# B&R Automation Studio project TD52 (part 102)

#### perm_par.var
```iecst
VAR
	tParaIntern : ParaHandler_typ; (*Connector type to perm_par*)
	tMM2ParaBase_ReadBack : MM2ParaBase_type; (*INTERNAL! V4.06 new readback structure for information from previous tasks*)
	bWriteDataObj : BOOL; (* TRUE=write data object module *)
	bDataObjLenErr : BOOL; (*Error occured in permem: data module size missmatch*)
	bCreateDataObj : BOOL; (* TRUE=create new data object *)
	bWriteOnce : BOOL; (* write permanent memory once *)
	DatObjCreate_01 : DatObjCreate; (* data object create *)
	DatObjInfoBak_02 : DatObjInfo; (* data object info *)
	DatObjDelete_01 : DatObjDelete; (* data object delete *)
	DatObjRead_01 : DatObjRead; (* data object read *)
	DatObjRead_02 : DatObjRead; (* manual initiated data object read *)
	DatObjWrite_01 : DatObjWrite; (* data object write *)
	DatObjDelete_02 : DatObjDelete; (* data object delete *)
	DatObjDelete_11 : DatObjDelete; (*Delete Backup File*)
	DatObjInfo_01 : DatObjInfo; (* data object info *)
	DatObjInfo_02 : DatObjInfo; (* data object info *)
	szModuleName : STRING[35]; (* module name of object *)
	szModuleNameBackup : STRING[35]; (* module name of posiibly created backup object *)
	DatObjCopy_01 : DatObjCopy;
	bCopyDataObj : BOOL;
	TON_WarnDelay : TON;
	TON_WritePMEM : TON; (* delay write permanent memory *)
	ulPMPointer : UDINT; (* adress of actual checksum value *)
	ulChecksum : UDINT; (* parameter checksum value *)
	pm_len : UDINT; (* permanent value lenght *)
	ulChecksumOld : UDINT; (* last vlaue of parameter checksum *)
	ulChkValue : UDINT; (* actual value of parameter pointer *)
	pm_id : UDINT; (* permanent value identifier *)
	pm_p : UDINT; (* permanent value pointer *)
	DatObjInfo_META : DatObjInfo;
	DatObjRead_META : DatObjRead;
	szMetaDataRaw : STRING[2000];
	szMetaData : ARRAY[0..4] OF STRING[35];
	szMetaDataVis : ARRAY[0..3] OF STRING[35];
	ssIndex : INT;
	ssCount : INT;
	ucMetaDataRaw : ARRAY[0..2000] OF USINT;
	ssCount2 : INT;
	szMetaDataFile : STRING[10];
	szText1 : STRING[20];
	pv_adr_IN_XX_tPB2MM : UDINT;
	pv_lng : UDINT;
	pv_lng_IN_XX_tPB2MM : UDINT;
	pv_lng_OUT_XX_tPB2MM : UDINT;
	szText2 : STRING[20];
	pv_adr_OUT_XX_tXX2PB : UDINT;
END_VAR
VAR CONSTANT
	ERR_NOERROR : UINT := 0;
END_VAR
VAR
	usPMWriteCnt : UINT;
	pm_Error : UDINT; (* permanent value error *) (* Deleted: pm : ParaMem_typ; permanent memory tags mathias, 22.8.11*)
	fun_Error : UDINT := 0; (*state > 0 = function error*)
	xLocalParaCheck : ParaCheckFUB; (*local function instance to check parameter values*)
	TON_ParaSetupOk : TON;
	bParaCheckSystemOk : BOOL;
	iDebug_ParaOkChecked : UDINT;
	bRestoreBackupDataObj : BOOL := FALSE;
	bRestoreDataObjContent : BOOL := FALSE;
	pm_id_backup : UDINT;
	pm_p_Backup : UDINT;
	DatObjCopy_02 : DatObjCopy;
	bDeleteBackupDataObj : BOOL := FALSE; (*Command to delete backup data module file on purpose*)
	bDebugPara : ARRAY[0..5] OF BOOL;
	ssIndex2 : INT;
	ssIndex3 : INT;
	ssIndex4 : INT;
	ssIndexVis : INT;
	szText : STRING[40];
	pv_adr_Para : UDINT;
	szParaSnippet : ARRAY[0..5] OF STRING[150];
	szParaIndex : STRING[10];
	slValue : DINT;
	iModuleDLD_ResetCount : INT;
	bDownloadDetected : BOOL;
	bFlagParaStructCopyWorking : BOOL; (*true, if cyclic para copying is active, 1 false cycle at every copy *)
	bStoreInitParaInDataObj : BOOL := FALSE;
	bTestflag : BOOL;
	bReadOutMETA_Once : BOOL;
	tParaCheck_iPvAdress : ARRAY[0..5] OF UDINT;
	tParaCheck_iPvLengt : ARRAY[0..5] OF UDINT;
	tParaCheck_rPvValue : ARRAY[0..5] OF REAL;
	tParaCheck_rRangeMIN : ARRAY[0..5] OF REAL;
	tParaCheck_rRangeMAX : ARRAY[0..5] OF REAL;
	tParaCheck_szPvName : ARRAY[0..5] OF STRING[35];
	ssFormatDetected : INT;
	szMetaDataPart : STRING[150];
	szFullTaskName : STRING[35];
	szFullMetaModuleName : STRING[35];
	debugLen : INT;
	debugSize : INT := 0;
	strcat_adr1 : UDINT;
	strcat_adr2 : UDINT;
	ssIndexTN : INT;
	bAlternate : BOOL;
	n : INT;
	iAlternateChecksum : DINT;
	iAlternateChecksumOld : DINT;
	ulDebugChkValue : ARRAY[0..999] OF UDINT;
	Adr1 : UDINT;
	Adr2 : UDINT;
	usPMWriteCntStepsize : UINT := 1; (*different step sizes to help debug*)
	usPMWriteCntXOR : UINT;
	usPMWriteCntAltSum : UINT;
	ulAdrPM : UDINT;
	usChkValuePM : USINT;
	ulAdrPara : UDINT;
	ulPara_len : UDINT;
	usChkValuePara : USINT;
	iDebugCountPMDifferences : DINT := 0;
	bEngineRunDetected : BOOL; (*detection status bit autocommand 100 /101  for engine run state*)
	ucMetaDataDebugInfoLine : ARRAY[0..24] OF STRING[80];
	ssIndexMand : INT := 0;
	szMetaDataMand : STRING[35];
	iMyErrorInfo_Autoreset : DINT; (*internal autoreset counter*)
	ssIndex_Version : INT; (*internal*)
	ssIndex_BU : INT; (*internal*)
	ssIndex_BU2 : INT; (*internal*)
END_VAR
```

### Program Logical/Generator/VisGC (IEC, version 4.09.0) - Visualization <-> Metamodule

#### VisGCCyclic.st
```iecst
(********************************************************************
VisGC	 			 General issues are handled here

This code is confidential and proprietary to the INNIO Company.
It may not be used in any form, or reproduced in any manner,
without written permission of the INNIO Company.
Copyright, INNIO Company, 2019

Customized modifications: -
------------------------

History:
-------
4.00.0	01.01.2013	ganguly		new
4.00.0	16.05.2014	lettenb.	cleanup
4.04.0	29.06.2016	lettenb.	tGen_T_In2 added, Dig142
4.05.0	30.11.2017	lettenb.	Q-management, unused MM2VIS-var removed
4.07.0	11.10.2018	lettenb.	Di: tU_Gen_Inc/Dec added for diagnosis
		29.04.2019	lettenb.	bU_Gen_Inc/Dec puls elongation for vis added(request requisition, mayer)
4.09.0	02.12.2019	lettenb.	ground failure counter added

Instructions for use: -
--------------------

Outstandings:
------------

*******************************************************************************)

PROGRAM _CYCLIC

	MM2VIS.bP_CosPCtr_Red_F_Hi     := OUT_GC.bP_Red_CosPCtr_F_Hi;
	MM2VIS.bP_CosPCtr_Red_F_Lo     := OUT_GC.bP_Red_CosPCtr_F_Lo;
	MM2VIS.bP_CosPCtr_Red_U_Hi     := OUT_GC.bP_Red_CosPCtr_U_Hi;
	MM2VIS.bP_CosPCtr_Red_U_Lo     := OUT_GC.bP_Red_CosPCtr_U_Lo;
	MM2VIS.rP_Gen_ppt              := rP_Gen_ppt;

	MM2VIS.rPF_CosPCtr_Set_Ctr13   := rPF_CosPCtr_Set_Ctr13;
	MM2VIS.rP_Red_CosPCtr_F        := rP_CosPCtr_F_Red;
	MM2VIS.rP_Red_CosPCtr_U        := rP_CosPCtr_U_Red;
	MM2VIS.rP_Red_CosPCtr_T        := rP_CosPCtr_T_Red;

	MM2VIS.rQ_CosPCtr_Set          := rQ_CosPCtr_Set;

	MM2VIS.rU_Gen_Exc              := OUT_GC.rU_Gen_Exc;

	MM2VIS.rT_Gen_Bear_A_Act       := IN_GC.tT_Gen_Bear_A_Act.Ai;
	MM2VIS.rT_Gen_Bear_B_Act       := IN_GC.tT_Gen_Bear_B_Act.Ai;
	MM2VIS.rT_Gen_Wind_Act_L1      := IN_GC.tT_Gen_Wind_Act_L1.Ai;
	MM2VIS.rT_Gen_Wind_Act_L2      := IN_GC.tT_Gen_Wind_Act_L2.Ai;
	MM2VIS.rT_Gen_Wind_Act_L3      := IN_GC.tT_Gen_Wind_Act_L3.Ai;
	MM2VIS.rT_Gen_Wind_Act         := IN_GC.tT_Gen_Wind.Ai;

	(* Oilskid *)
	MM2VIS.bOilSkid_PumpLP_Dem 		:= OUT_GC.tOilSkid_PumpLP.Do;
	MM2VIS.bOilSkid_PumpHP_Dem		:= OUT_GC.tOilSkid_PumpHP.Do OR OUT_GC.tOilSkid_PumpHP_UPS.Do;
	MM2VIS.bOilSkid_PumpC_Dem 		:= OUT_GC.tOilSkid_PumpC.Do;
	MM2VIS.bOilSkid_Fan_Dem 		:= OUT_GC.tOilSkid_Fan.Do;
	MM2VIS.bOilSkid_Heater_Dem 		:= OUT_GC.tOilSkid_Heater.Do;
	MM2VIS.rLev_OilSkid_Tank		:= IN_GC.tLev_OilSkid_Tank.Ai;
	MM2VIS.rT_OilSkid_Tank			:= IN_GC.tT_OilSkid_Tank.Ai;
	MM2VIS.rPr_OilSkid_HP_NDE		:= IN_GC.tPr_OilSkid_HP_NDE.Ai;
	MM2VIS.rPr_OilSkid_HP_DE		:= IN_GC.tPr_OilSkid_HP_DE.Ai;
	MM2VIS.rFlow_OilSkid_DE			:= IN_GC.tFlow_OilSkid_DE.Ai;
	MM2VIS.rFlow_OilSkid_NDE		:= IN_GC.tFlow_OilSkid_NDE.Ai;
	MM2VIS.rT_OilSkid_Supply		:= IN_GC.tT_OilSkid_Supply.Ai;

	MM2VIS.rF_GenBear_DE1			:= IN_GC.tF_GenBear_DE1.Ai;
	MM2VIS.rF_GenBear_DE2			:= IN_GC.tF_GenBear_DE2.Ai;
	MM2VIS.rF_GenBear_NDE1			:= IN_GC.tF_GenBear_NDE1.Ai;
	MM2VIS.rF_GenBear_NDE2			:= IN_GC.tF_GenBear_NDE2.Ai;

	MM2VIS.rGen_T_In				:= IN_GC.tGen_T_In.Ai;
	MM2VIS.rGen_T_In2				:= IN_GC.tGen_T_In2.Ai;
	MM2VIS.rT_GenAirOut				:= IN_GC.tT_GenAirOut.Ai;

	xTP_U_Gen_Inc(IN:= EDGEPOS(IN_GC.tU_Gen_Inc.Di OR IN_GC.tU_Adj_Plus.Di), PT:= T#2s);(* DI voltage adjustment external (increasing)*)
	MM2VIS.bU_Gen_Inc				:= xTP_U_Gen_Inc.Q;

	xTP_U_Gen_Dec(IN:= EDGEPOS(IN_GC.tU_Gen_Dec.Di OR IN_GC.tU_Adj_Minus.Di), PT:= T#2s);(* DI voltage adjustment external (decreasing)*)
	MM2VIS.bU_Gen_Dec				:= xTP_U_Gen_Dec.Q;

	MM2VIS.bCntGndFail_Visible 		:= IN_GC.tGndFaultW.GoodQual; (* counter visibility *)

END_PROGRAM
```

#### VisGC.var
```iecst
VAR
  	xTP_U_Gen_Inc : TP;
  	xTP_U_Gen_Dec : TP;
END_VAR

VAR CONSTANT

END_VAR
```

### Program Logical/Generator/MMUEarthFault (IEC) - MMU Earth Fault detection

#### MMUEarthFaultCyclic.st - Program
```iecst
(********************************************************************
MMUEarthFault	 			 Earth Fault Detection via MMU Signals

This code is confidential and proprietary to the INNIO Company.
It may not be used in any form, or reproduced in any manner,
without written permission of the INNIO Company.
Copyright, INNIO Company, 2023

Customized modifications: -
------------------------

History:
-------
4.13.0	29.06.2023	Perktold	new

Instructions for use: -
--------------------

Outstandings:
------------

*******************************************************************************)
PROGRAM _CYCLIC

IF Para.rU_Gen_Nom[1] <> 0 THEN

	//Activate monitoring 2s after at least one Ph-Ph-Voltage exceeds 50% nominal voltage
	xTON_MonAct(IN := (MAX(IN_GC.tU_L1L2[1].Ai, IN_GC.tU_L2L3[1].Ai, IN_GC.tU_L3L1[1].Ai) > (Para.rU_Gen_Nom[1] * 0.5)), PT := T#2s);

	IF xTON_MonAct.Q THEN

		//Read pos. zero crossing time stamps and convert to [ms]
		rTimeStamp_PosZeroCrossing_UGen1 := DINT_TO_REAL(IN_GC.iTimeStamp_PosZeroCrossing_UGen1) / 4096000;	(* [ms] *)
		rTimeStamp_PosZeroCrossing_UGen2 := DINT_TO_REAL(IN_GC.iTimeStamp_PosZeroCrossing_UGen2) / 4096000;	(* [ms] *)
		rTimeStamp_PosZeroCrossing_UGen3 := DINT_TO_REAL(IN_GC.iTimeStamp_PosZeroCrossing_UGen3) / 4096000;	(* [ms] *)

		//Correct values for easy comparison if values overrun the DINT the negatve values get corrected by 1048.5759ms (total DINT range)
		iNumNeg	:= 0;
		IF ABS(rTimeStamp_PosZeroCrossing_UGen1) > 200 AND ABS(rTimeStamp_PosZeroCrossing_UGen2) > 200 AND ABS(rTimeStamp_PosZeroCrossing_UGen3) > 200 THEN
			IF rTimeStamp_PosZeroCrossing_UGen1 < 0.0 THEN	iNumNeg	:= iNumNeg + 1;	END_IF;
			IF rTimeStamp_PosZeroCrossing_UGen2 < 0.0 THEN	iNumNeg	:= iNumNeg + 1;	END_IF;
			IF rTimeStamp_PosZeroCrossing_UGen3 < 0.0 THEN	iNumNeg	:= iNumNeg + 1;	END_IF;

			IF (iNumNeg = 1) OR (iNumNeg = 2) THEN
				IF rTimeStamp_PosZeroCrossing_UGen1 < 0.0 THEN
					rTimeStamp_Calc_UGen1	:= rTimeStamp_PosZeroCrossing_UGen1 + 1048.57599975586;	(* [ms] *)
				ELSE
					rTimeStamp_Calc_UGen1	:= rTimeStamp_PosZeroCrossing_UGen1;					(* [ms] *)
				END_IF;

				IF rTimeStamp_PosZeroCrossing_UGen2 < 0.0 THEN
					rTimeStamp_Calc_UGen2	:= rTimeStamp_PosZeroCrossing_UGen2 + 1048.57599975586;	(* [ms] *)
				ELSE
					rTimeStamp_Calc_UGen2	:= rTimeStamp_PosZeroCrossing_UGen2;					(* [ms] *)
				END_IF;

				IF rTimeStamp_PosZeroCrossing_UGen3 < 0.0 THEN
					rTimeStamp_Calc_UGen3	:= rTimeStamp_PosZeroCrossing_UGen3 + 1048.57599975586;	(* [ms] *)
				ELSE
					rTimeStamp_Calc_UGen3	:= rTimeStamp_PosZeroCrossing_UGen3;					(* [ms] *)
				END_IF;
			ELSE
				rTimeStamp_Calc_UGen1	:= rTimeStamp_PosZeroCrossing_UGen1;						(* [ms] *)
				rTimeStamp_Calc_UGen2	:= rTimeStamp_PosZeroCrossing_UGen2;						(* [ms] *)
				rTimeStamp_Calc_UGen3	:= rTimeStamp_PosZeroCrossing_UGen3;						(* [ms] *)
			END_IF;
		ELSE
			rTimeStamp_Calc_UGen1	:= rTimeStamp_PosZeroCrossing_UGen1;							(* [ms] *)
			rTimeStamp_Calc_UGen2	:= rTimeStamp_PosZeroCrossing_UGen2;							(* [ms] *)
			rTimeStamp_Calc_UGen3	:= rTimeStamp_PosZeroCrossing_UGen3;							(* [ms] *)
		END_IF;

		//get the three values in the right order
		rTimeStamp_max	:= MAX(rTimeStamp_Calc_UGen1, rTimeStamp_Calc_UGen2, rTimeStamp_Calc_UGen3);
		rTimeStamp_min	:= MIN(rTimeStamp_Calc_UGen1, rTimeStamp_Calc_UGen2, rTimeStamp_Calc_UGen3);

		IF (rTimeStamp_Calc_UGen1 <> rTimeStamp_max) AND (rTimeStamp_Calc_UGen1 <> rTimeStamp_min) THEN
			rTimeStamp_mid	:= rTimeStamp_Calc_UGen1;
		ELSIF (rTimeStamp_Calc_UGen2 <> rTimeStamp_max) AND (rTimeStamp_Calc_UGen2 <> rTimeStamp_min) THEN
			rTimeStamp_mid	:= rTimeStamp_Calc_UGen2;
		ELSE
			rTimeStamp_mid	:= rTimeStamp_Calc_UGen3;
		END_IF;

		//Calculate time difference beween the time stamps
		rDelta_1 := rTimeStamp_mid - rTimeStamp_min;							(* [ms] *)
		rDelta_2 := rTimeStamp_max - rTimeStamp_mid;							(* [ms] *)

		rTPeriodTime	:= 1.0 / LIMIT(0.1, IN_GC.tF_MMD[1].Ai, 70.0) * 1000;	(* [ms] *)
		//convert to angle difference
		rDAng_1			:= rDelta_1 / rTPeriodTime * 360.0;						(* [Deg] *)
		rDAng_2			:= rDelta_2 / rTPeriodTime * 360.0;						(* [Deg] *)

		//Check if the values are 120[Deg] +- rDAng_Dev
		IF (rDAng_1 > (120.0 - rDAng_Dev)) AND (rDAng_1 < (120.0 + rDAng_Dev)) THEN
			bDANg_1_ok	:= TRUE;
		ELSE
			bDANg_1_ok	:= FALSE;
		END_IF

		IF (rDAng_2 > (120.0 - rDAng_Dev)) AND (rDAng_2 < (120.0 + rDAng_Dev)) THEN
			bDANg_2_ok	:= TRUE;
		ELSE
			bDANg_2_ok	:= FALSE;
		END_IF

		//trigger warning and trip if at least on value stays out of range for a vertain time
		xTON_warning(IN := ((NOT bDANg_1_ok OR NOT bDANg_2_ok) AND Para.bMMDGroundFaultMonAct AND (Para.tTi_MMDGroundFaultWarning > T#0ms)), PT := Para.tTi_MMDGroundFaultWarning);
		xTON_trip(IN 	:= ((NOT bDANg_1_ok OR NOT bDANg_2_ok) AND Para.bMMDGroundFaultMonAct AND (Para.tTi_MMDGroundFaultTrip > T#0ms)), PT := Para.tTi_MMDGroundFaultTrip);

		bMsg9372_set			:= xTON_warning.Q;		(*W9372 Multi measurement device: Earth failure generator*)
		bMsg2373_set			:= xTON_trip.Q;			(*A2373 Multi measurement device: Earth failure generator*)
	ELSE
		bMsg9372_set			:= FALSE;
		bMsg2373_set			:= FALSE;
		xTON_warning(IN := FALSE, PT := Para.tTi_MMDGroundFaultWarning);
		xTON_trip(IN 	:= FALSE, PT := Para.tTi_MMDGroundFaultTrip);
	END_IF;
ELSE
	bMsg9372_set	:= FALSE;
	bMsg2373_set	:= FALSE;
	xTON_warning(IN	:= FALSE, PT := Para.tTi_MMDGroundFaultWarning);
	xTON_trip(IN 	:= FALSE, PT := Para.tTi_MMDGroundFaultTrip);
	xTON_MonAct(IN 	:= FALSE, PT := T#2s);
END_IF;

END_PROGRAM
```

#### MMUEarthFault.var - Variables
```iecst
VAR
	rTimeStamp_PosZeroCrossing_UGen1 : REAL := 0.0; (*[ms]*)
	rTimeStamp_PosZeroCrossing_UGen2 : REAL := 0.0; (*[ms]*)
	rTimeStamp_PosZeroCrossing_UGen3 : REAL := 0.0; (*[ms]*)
	rTPeriodTime : REAL; (*[ms]*)
	rTimeStamp_Calc_UGen1 : REAL := 0.0;
	rTimeStamp_Calc_UGen2 : REAL := 0.0;
	rTimeStamp_Calc_UGen3 : REAL := 0.0;
	rTimeStamp_max : REAL := 0.0;
	rTimeStamp_min : REAL := 0.0;
	rTimeStamp_mid : REAL := 0.0;
	iNumNeg : INT := 0;
	rDelta_1 : REAL := 0.0;
	rDelta_2 : REAL := 0.0;
	rDAng_1 : REAL := 0.0;
	rDAng_2 : REAL := 0.0;
	rDAng_Dev : REAL := 10.0;
	bDANg_1_ok : BOOL := 0;
	bDANg_2_ok : BOOL := 0;
	xTON_warning : TON;
	xTON_trip : TON;
	xTON_MonAct : TON;
END_VAR
```

### Package Logical/GasMeteringUnit - GD: Gas Metering Unit Device

### Data object Logical/GasMeteringUnit/META_GD (Simple) - Simple data object.

#### META_GD.dat
```
; *******************************************************************************
; AGGR: Module Meta Data (data module)
;
; This code is confidential and proprietary to the INNIO Company.
; It may not be used in any form, or reproduced in any manner, without the express
; written permission of the INNIO Company.
; Copyright, INNIO Company, 2023
;
; Customized modifications: -
; ------------------------
;
; History:
; -------
; V3.99	06-03-2013	Weitzer, generated for modular software
; V4.00 11-09-2013  pankajrodey, updated file with relevant information
; V4.01 18-10-2013  Zengerer   typo corr., NO duplicate para Chk entries!
; 		08-05-2014  Weitzer, switch to CAN interface identifier from HAL_IO
;							 "hard code" missing parameters
; V4.04.00.00	04-07-2016	Gwiggner,	Bugfix: Tecjet Monitoring
; V4.04.00.00	05-08-2016	Gwiggner,	Bugfix: Mapping bDualTJ
; V4.04.00.00	28-10-2016	Gwiggner,	Bugfix: correction interpolation of gas density
; V4.05.00.00	27.07.2017	Messner,	CAN Diagnosis Picture added
; V4.05.01.00	05.04.2018	Perktold,	GMU - Monitoring Delay for TJs increased from 5 to 7s
; V4.11.00.00	15.11.2021	Perktold,	defined ucTecNr as local variable, correction REAL_TO_USINT -> INT_TO_USINT, A3093 DGS
; V4.12.00.00	13.12.2022	Gwiggner,	GMU self diagnosis
; V4.12.00.00	22.01.2023	Zuschnig,	Interpolation od gas density done in EC module
; V4.13.00.00	16.11.2022	Gwiggner,	adaption for W3213 & B3249
;
; Instructions for use:
; --------------------
; make only changes at the version numbers
;
; Outstandings:
; ------------
;
; *******************************************************************************
;
"<META>"
;
; Module ID
"<MODUL>GD</MODUL>"
;
; Module Version (xx.yy.zz.cc)
"<VERSION>04.13.00.00</VERSION>"
;
; Module Basisupdate Version BU (00-99)
"<BASISUPDATE_VERSION>00</BASISUPDATE_VERSION>"
;
; Optional: specify order number for limitated module usage
"<ORDER></ORDER>" ;<!--(optional for restricted customizations; missing statement makes module valid for all orders)-->
;
; Parameter Check <PARAn Name='aAbcdef' MIN='xxx' MAX='yyy' />  (watch for correct spacings and apostrophs!)
"<PARAMETER_CHK>"
"<PARA1 Name='iEng_Motortype' MIN='208' MAX='920' />"
"<PARA2 Name='iN_GMU_Devices' MIN='0' MAX='5' />"
"<PARA3 Name='usGasDensN[1]' MIN='200' MAX='2500' />"
"<PARA4 />"
"<PARA5 />"
"</PARAMETER_CHK>"
;
; <--Permanent Datamodule Filenames:  NAME ist ohne Dateiendung einzutragen; Nur für Counter und interne Parameter verwenden-->
"<DATAMODULES>" ;<!-- optional; mehrere DATAMODULES erlaubt-->
"	<DATAMODULE>par_GD</DATAMODULE>"
"</DATAMODULES>"
;
; Dependencies Modules (MMxx.yy.zz.cc)
"<DEPENDENCIES>"
"	<DEPENDENCY MODULE='AB' VERSION='04.00.00.00' />"
"	<DEPENDENCY MODULE='PB' VERSION='04.00.00.00' />"
"	<DEPENDENCY MODULE='GT' VERSION='04.12.00.00' />"
"	<DEPENDENCY MODULE='OP' VERSION='04.00.00.00' />"
"	<DEPENDENCY MODULE='HA' VERSION='04.05.00.00' />"
"	<DEPENDENCY MODULE='EC' VERSION='04.12.00.00' />"
"   <DEPENDENCY VISVERSION='02.06.00.00' />"			; Dependencies Visualization
"</DEPENDENCIES>"
;
; Module function description
"<MODULEFUNCTION>" ;<!-- short overview documentation of module function; add reference to detailed information, if available-->
"	<General>	"
"	GD Module for the TecJet(tm) valve actuator - an integrated and digitally compensated control valve and actuator system"
" 	for regulating and metering the flow of gas "
"	</General>	"
""
"	<F1 Name='Gas metering' LastModified='4.0.0.0'>"
"	These paramaeters of the Air-Fuel mixture are measured by the module:	"
"	Valve differential pressure, Valve position, Gas Temperature, Running hours, Software version, Gas pressure	"
"	</F1>"
"	<F2 Name='Errors and alarms' LastModified='4.0.0.0'>"
"	Errors in the Tecjet module are sent by this module to the controller	"
"	</F2>"
"	<F3 Name='enter name of main function 3 here' LastModified='4.0.0.0'>"
"	Enter function 3 description for module here.	"
"	</F3>"
""
"	<Info>"
"	V4.04.00.00	Bugfix: Tecjet Monitoring	"
"   V4.04.00.00	Bugfix: Mapping bDualTJ	"
"   V4.04.00.00	Bugfix: correction interpolation of gas density	"
"	</Info>"
""
"	<Customized LastModified='4.0.0.0'>	"
"	- Nothing "
"	</Customized>	"
""
"</MODULEFUNCTION>"
;
"</META>"
```

### module_GD.typ - Package data types
```iecst
(*******************************************************************************
	module_GMU : Type definitions for the GMU module

	This code is confidential and proprietary to the INNIO Company.
	It may not be used in any form, or reproduced in any manner, without the express
	written permission of the INNIO Company.
	Copyright, INNIO Company, 2019

	- calcualtion of different gas inject valve concerning parameters for gas sort 0
	- send parameter to gas inject valve
	- handling gas inject valve communication problem
	- read software version, operating hours, and gas inject valve status
	- check gas inject valve software version

	Customized modifications: -
	------------------------

	History:
	-------

	V3.99.0 07-04-2012  pankajrodey	,  Added new version for Modular software
	V3.99.1 28-08-2012  pankajrodey	,  Added structures for MM2VIS ans VIS2MM

	Instructions for use:
	--------------------

	Outstandings:
	------------
	*******************************************************************************)

TYPE
	IN_GD_struct : 	STRUCT
		tPB2MM : ParaBase2MM_type; (*parameter setup ok*) (*OldName: FGDRPS; Cycle: 5*)
		tGV1_Open : HALioDo_Type; (*DO: open gas valve 1*) (*OldName: GASV1; Cycle: 5*)
		tAB2GD : AmmBase2MM;
		tGV2_Open : HALioDo_Type; (*DO: open gas valve 2*) (*OldName: GASV2; Cycle: 5*)
		rP_Act_Norm_Filt : REAL; (*actual power related to rP_Nom [%] filtered T=1s*) (*OldName: P_IST_PROM; Cycle: 5*)
		iCANIdent : UDINT; (*CAN open status from CAN module*) (*OldName: new; Cycle: 5*)
		iSt_OpMode : UDINT; (* engine operation mode *) (*OldName: new; Cycle: 5*)
		ulGasFlowN : ARRAY[0..4]OF UDINT; (* setpoint gasflow one gas inject v *) (*OldName: ulGasFlowN; Cycle: 5*)
		iIdx_Gtyp_Dem : INT; (* actual gassort 1..4 *)
		bSimWinMOD_Active : BOOL;
		ulMonGasFlow : ARRAY[0..4]OF UDINT; (* minimum flow for monitoring *) (* OldName: ulMonGasFlow; Cycle: 2 *)
		bDualTJ : BOOL; (*Gas mixing with two TecJet´s*) (*OldName: bDualTJ; Cycle:5*)
		bDualTJ_TC2 : BOOL; (*Gas mixing with two TecJet´s*) (*OldName: bDualTJ; Cycle:2*)
		bLR_GasStop : BOOL; (*close gas valve to react on a load rejection by the GCB and force  actuators (open CBP, close TV)*)
		rGT_QualMix_1_2 : REAL; (*Mixture ratio between gas 1 and 2 [%]*) (*OldName: 	ssMisch1_2; Cycle: ; *)
		bCANCntReset : BOOL; (* CAN error counter value reset *) (*OldName: bCANCounterReset; Cycle:5;*)
		usGasDensN : ARRAY[0..4]OF UINT; (*Nominal gas density for usGasDensN*)
	END_STRUCT;
	OUT_GD_struct : 	STRUCT
		rGMU_Pr_DiffGas : ARRAY[0..4]OF REAL; (*Differential Pressure over device [mbar*10]*) (*OldName: ulGasFlowN; Cycle: 5*)
		rGMU_Pos_Valve_Rad : ARRAY[0..4]OF REAL; (*Valve Position [rad *10]*) (*OldName: ssValvePos; Cycle: 5*)
		rGMU_Pos_Valve_Prom : ARRAY[0..4]OF REAL; (*Valve Position [%o]*) (*OldName: ssTJPos; Cycle: 5*)
		rGMU_Pr_FuelGas : ARRAY[0..4]OF REAL; (*Fuel Gas Pressure at device inlet [mbar*10]*) (*OldName: ssGasPress; Cycle: 5*)
		rGMU_T_FuelGas : ARRAY[0..4]OF REAL; (*Fuel Gas Temperature at device inlet [°C *10]*) (*OldName: ssGasTemp; Cycle: 5*)
		rGMU_Q_FuelGas : ARRAY[0..4]OF REAL; (*Fuel Gas Amount denormalized [l/s*1000]*) (*OldName: slGasFlow; Cycle: 5*)
		rGMU_D_FuelGas : ARRAY[0..4]OF REAL; (*Fuel Gas Density denormalized [kg/m3*1000]*) (*OldName: ssGasDens; Cycle: 5*)
		rGMU_N_RunningHours : ARRAY[0..4]OF REAL; (*Running hours of device [hours]*) (*OldName: usRHourTJ; Cycle: 5*)
		rGMU_S_Status : ARRAY[0..4]OF REAL; (*Status of device [-]*) (*OldName: usStateTJ; Cycle: 5*)
		tGD2AB : MM2AmmBase; (* *) (*OldName: new; Cycle: 5*)
		rGMU_Vers_SW : ARRAY[0..4]OF REAL; (*Firmware version*) (*OldName: usSWTecJet; Cycle: 5*)
		tGasMeteringUnit_CanGo : CanDeviceGo; (* *) (*OldName: new; Cycle: 5*)
		tGD2PB : MM2ParaBase_type; (* *) (*OldName: new; Cycle: 5*)
		iTecErrCntMax : ARRAY[0..4]OF USINT; (* max value for wrong gas flow trans *)
		iTecErrCnt : ARRAY[0..4]OF USINT; (* counter for wrong gas flow transm. *)
		iTecJetCommErrCount : USINT; (* timeout counter for comm. error *)
		tE_TEC : ARRAY[0..4]OF _tEventTEC; (* CAN events gas inject valve param. *)
		sGMU_Num_HWP : ARRAY[0..4]OF STRING[10]; (*Hardware part number of device*) (*OldName: new; Cycle: 5*)
		iGMU_Num_Ser : ARRAY[0..4]OF UDINT; (*serial number of device*) (*OldName: new; Cycle: 5*)
	END_STRUCT;
	Para_struct : 	STRUCT
		iN_GMU_CAN : INT; (*Para: CAN node number of first device*) (*OldName: TecJet_Node; Cycle: 5*)
		iN_GMU_Devices : INT; (*PARA [11352]: Number of installed gas metering devices*) (*OldName: ucNrOfTJ; Cycle: 5*)
		usGasDensN : ARRAY[0..4]OF INT; (*Para: Nominal gas density *) (*OldName: usGasDensN; Cycle: 5*)
		rConst_GMU_Gas : REAL; (*Para: gas constant (default:=1300)*) (*OldName: usWobbeRef; Cycle: 5*)
		bGMU_ResetRunningHours : BOOL; (*Para: TRUE = reset running hours*) (*OldName: bReRunHour; Cycle: 5*)
		rPr_GMU_DiffMinimum : REAL; (*Para: Minimal allowed delta pressure over device [mbar] (default:= -20)*) (*OldName: ssMinDP; Cycle: 5*)
		rPr_GMU_DiffMaximum : REAL; (*Para: Maximal allowed delta pressure over device [mbar] (default:= 500)*) (*OldName: ssMaxDP; Cycle: 5*)
		rPr_GMU_Minimum : REAL; (*Para : Minimal allowed inlet fuel gas pressure [mbar] (default:= 500)*) (*OldName: ssMinPress; Cycle: 5*)
		rPr_GMU_Maximum : REAL; (*Para: Maximal allowed inelt fuel gas pressure [mbar] (default:= 1600)*) (*OldName: ssMaxPress; Cycle: 5*)
		rT_GMU_Minimum : REAL; (*Para: Minimal allowed fuel gas temperature [°C] (default:= -20)*) (*OldName: ssTempMin; Cycle: 5*)
		rT_GMU_Maximum : REAL; (*Para: Maximal allowed fuel gas temperature [°C] (default:= 90)*) (*OldName: ssTempMax; Cycle: 5*)
		iEng_Motortype : INT;
		bEng_Act_H2 : BOOL; (* PARA [tbd]: H2 engine active *)
	END_STRUCT;
	MM2VIS_struct : 	STRUCT
		bMsg3093 : BOOL; (*3093*) (*OldName: TJ_Can; Cycle: 5*)
		bMsg3241 : BOOL; (*3241: Operating message tecjet CAN failure*) (*OldName: TJ_CAN_B; Cycle: 5*)
		iMsg3241 : INT; (*Error number tecjet CAN failure*) (*OldName: ucTJ_CAN; Cycle: 5*)
		bMsg3094 : BOOL; (*3094*) (*OldName: TJ_Softw; Cycle: 5*)
		bMsg3242 : BOOL; (*Operating message wrong Software version*) (*OldName: TJ_SOFTW_B; Cycle: 5*)
		iMsg3242 : INT; (*Error number wrong Software version*) (*OldName: ucTJ_SOFTW; Cycle: 5*)
		bMsg3095 : BOOL; (*3095*) (*OldName : TJ_GasT; Cycle : 5*)
		bMsg3243 : BOOL; (*Operating message : Gas temperature*) (*OldName : TJ_GAST_B; Cycle : 5*)
		iMsg3243 : INT; (*Error number : Gas Temperature*) (*OldName : ucTJ_GAST; Cycle : 5*)
		bMsg3096 : BOOL; (*3096*) (*OldName: TJ_GasD; Cycle: 5*)
		bMsg3244 : BOOL; (*Operating message : Gas differential pressure*) (*OldName : TJ_GASD_B; Cycle : 5*)
		iMsg3244 : INT; (*Error number : Gas differential pressure*) (*OldName : ucTJ_GASD; Cycle : 5*)
		bMsg3097 : BOOL; (*3097*) (*OldName: TJ_Int; Cycle: 5*)
		bMsg3245 : BOOL; (*Operating message : TECJET internal error*) (*OldName : TJ_INT_B; Cycle : 5*)
		iMsg3245 : INT; (*Error nmber : TECJET internal error*) (*OldName : ucTJ_INT; Cycle : 5*)
		bMsg3098 : BOOL; (*3098*) (*OldName: TJ_Mech; Cycle: 5*)
		bMsg3246 : BOOL; (*Operating message : TECTET Mechanical failure*) (*OldName : TJ_MECH_B; Cycle : 5*)
		iMsg3246 : INT; (*Error number : TECTET Mechanical failure*) (*OldName : ucTJ_MECH; Cycle : 5*)
		bMsg3213 : BOOL; (*3213*) (*OldName: TJ_GasN; Cycle: 5*)
		bMsg3249 : BOOL; (*Operating message : check gas inject valve gas flow not reached*) (*OldNmae : TJ_GASN_B; Cyclic : 5*)
		iMsg3249 : INT; (*Error number : check gas inject valve gas flow not reached*) (*OldName : ucTJ_GASN; Cyclic : 5*)
		rGMU_Pr_DiffGas : ARRAY[0..4]OF REAL; (*Differential Pressure over device [mbar*10]*) (*OldName: ssDPress; Cycle: 5*)
		rGMU_Pos_Valve_Rad : ARRAY[0..4]OF REAL; (*Valve Position [rad *10]*) (*OldName: ssValvePos; Cycle: 5*)
		rGMU_Pos_Valve_Prom : ARRAY[0..4]OF REAL; (*Valve Position [%o]*) (*OldName: ssTJPos; Cycle: 5*)
		rGMU_Pr_FuelGas : ARRAY[0..4]OF REAL; (*Fuel Gas Pressure at device inlet [mbar*10]*) (*OldName: ssGasPress; Cycle: 5*)
		rGMU_T_FuelGas : ARRAY[0..4]OF REAL; (*Fuel Gas Temperature at device inlet [°C *10]*) (*OldName: ssGasTemp; Cycle: 5*)
		rGMU_Q_FuelGas : ARRAY[0..4]OF REAL; (*Fuel Gas Amount denormalized [l/s*1000]*) (*OldName: slGasFlow; Cycle: 5*)
		rGMU_D_FuelGas : ARRAY[0..4]OF REAL; (*Fuel Gas Density denormalized [kg/m3*1000]*) (* OldName: ssGasDens; Cycle: 5*)
		rGMU_N_RunningHours : ARRAY[0..4]OF REAL; (*Running hours of device [hours]*) (*OldName: usRHourTJ; Cycle: 5*)
		rGMU_S_Status : ARRAY[0..4]OF REAL; (*Status of device [-]*) (*OldName: usStateTJ; Cycle: 5*)
		rGMU_Vers_SW : ARRAY[0..4]OF REAL; (*Firmware version*) (*OldName: usSWTecJet; Cycle: 5*)
		iCMSmain_TecJet_status : INT; (* TecJet CAN Module Main CMS Status *)
		iCMSinit_TecJet_status : INT; (* TecJet CAN Module CMS Init Status *)
		bFlow_GMU_Down : ARRAY[0..4]OF BOOL; (* zero flow detected *)
		bPr_Diff_GMU_Down : ARRAY[0..4]OF BOOL; (* zero flow detected *)
		bT_EU_GMU_HiHi : ARRAY[0..4]OF BOOL; (* Electronics temperature high *)
		bPos_GMU_Err : ARRAY[0..4]OF BOOL; (* Valve position error *)
		bFlow_GMU_Min : ARRAY[0..4]OF BOOL; (* flow not reached *)
		bValS_GMU_Ok : ARRAY[0..4]OF BOOL; (* Overall status ok *)
		bPr_GMU_HiHi : ARRAY[0..4]OF BOOL; (* fuel gas pressure high limit *)
		bPr_Diff_GMU_HiHi : ARRAY[0..4]OF BOOL; (* delta pressure high limit *)
		bT_GMU_HiHi : ARRAY[0..4]OF BOOL; (* fuel gas temp. high limit *)
		bU_GMU_HiHi : ARRAY[0..4]OF BOOL; (* Input voltage high limit *)
		bPr_GMU_LoLo : ARRAY[0..4]OF BOOL; (* fuel gas pressure low limit *)
		bPr_Diff_GMU_LoLo : ARRAY[0..4]OF BOOL; (* delta pressure low limit *)
		bT_GMU_LoLo : ARRAY[0..4]OF BOOL; (* fuel gas temp. low limit	*)
		bU_GMU_LoLo : ARRAY[0..4]OF BOOL; (* Input voltage low limit *)
		bInt_GMU_Err : ARRAY[0..4]OF BOOL; (* gas inject internal failure *)
		bMech_GMU_Err : ARRAY[0..4]OF BOOL; (* gas inject closed due to error - malfunction	*)
		bFlow_GMU_SetErr : ARRAY[0..4]OF BOOL; (* CAN flow demand failed *)
		sGMU_Num_HWP : ARRAY[0..4]OF STRING[10]; (* Tecjet hardware number*) (*OldName: usRHourTJ; Cycle: 5*)
		iGMU_Num_Ser : ARRAY[0..4]OF UDINT; (* Tecjet serial number*) (*OldName: usRHourTJ; Cycle: 5*)
		bGMU_SelfDiagnosis_ena : BOOL; (* Show Self Diagnosis Table on HMI *)
	END_STRUCT;
	CanDeviceGo : 	STRUCT
		CANDevGo : ARRAY[0..1]OF USINT;
		ECANDevGo : USINT;
	END_STRUCT;
	_tEventTEC : 	STRUCT
		Conf : ARRAY[0..8]OF USINT;
		Data : ARRAY[0..5]OF USINT;
		Contr : ARRAY[0..1]OF USINT;
		Status : ARRAY[0..5]OF USINT;
	END_STRUCT;
	_TecJetError : 	STRUCT
		ucError : ARRAY[0..7]OF USINT;
	END_STRUCT;
END_TYPE
```

### module_GD.var - Package variables
```iecst
(*******************************************************************************
	module_GMU : Module level global variables for the GMU module

	This code is confidential and proprietary to the INNIO Company.
	It may not be used in any form, or reproduced in any manner, without the express
	written permission of the INNIO Company.
	Copyright, INNIO Company, 2019

	- calcualtion of different gas inject valve concerning parameters for gas sort 0
	- send parameter to gas inject valve
	- handling gas inject valve communication problem
	- read software version, operating hours, and gas inject valve status
	- check gas inject valve software version

	Customized modifications: -
	------------------------

	History:
	-------

	V3.99.0 07-04-2012  pankajrodey	,  Added new version for Modular software
	V3.99.1 28-08-2012  pankajrodey	,  Added structures for MM2VIS ans VIS2MM
	V3.99.1 27-11-2013  pankajrodey	,  Deleted variables to remove compilation warning

	Instructions for use:
	--------------------

	Outstandings:
	------------
	*******************************************************************************)
VAR
	pm : Para_struct;
	Para : Para_struct;
	ParaFactoryDefault : Para_struct := (0);
	OUT_GD : OUT_GD_struct := (0);
	IN_GD : IN_GD_struct := (0);
	bSendParTecJet : BOOL; (* TJ Send Parameter to TecJet *)
	gasart : USINT; (* actual gassort 0 to 4 *)
	usGasDensN : ARRAY[0..4] OF UINT; (* nominal gas density *)
	ucNrTJCommErr : USINT; (* number of TJ valve comm. problem *)
	TecJet_ID : USINT; (* TecJet CAN-ID number *)
	bTecJetFlowErr : BOOL; (* TRUE=wrong transmission of gasflow *)
	ucTecJetCommErrCount : USINT; (* timeout counter for comm. error *)
	CANDevGo : ARRAY[0..1] OF USINT; (* startup parameter for CAN devices *)
	ECANDevGo : USINT; (* event startup parameter CAN device *)
	usSWTecJet : ARRAY[0..4] OF UINT; (* software version of all TecJet´s *)
	usWobbeRef : UINT; (* reference wobbe index TecJet *)
	bReRunHour : INT; (* set operating hour gas inject v. *)
	ssMinDP : INT; (* gas difference pressure minimum *)
	ssMaxDP : INT; (* gas difference pressure max. Tec *)
	ssMinPress : INT; (* gas pressure minimum TecJet *)
	ssMaxPress : INT; (* gas pressure maximum TecJet *)
	ssTempMin : INT; (* gastemperature minimum TecJet *)
	ssTempMax : INT; (* gas temperature maximum TecJet *)
	TJ_Can : ARRAY[0..4] OF BOOL; (* TJ CAN communication error *)
	ssDPress : ARRAY[0..4] OF INT; (* actual gas diffrence pressure *)
	ssValvePos : ARRAY[0..4] OF INT; (* actual valve position gas inject v *)
	ssGasPress : ARRAY[0..4] OF INT; (* actual gas pressure gas inject  v. *)
	ssGasTemp : ARRAY[0..4] OF INT; (* actual gas temp. gas inject valves *)
	slGasFlow : ARRAY[0..4] OF DINT; (* actual gas flow gas inject valves *)
	ssGasDens : ARRAY[0..4] OF INT; (* actual gas density gas inject valv *)
	usRHourTJ : ARRAY[0..4] OF UINT; (* running hour each gas inject valve *)
	usStateTJ : ARRAY[0..4] OF UINT; (* status of each gas inject valve *)
	usGasDens : ARRAY[0..4] OF UINT; (* actual gas density *)
	TJ_SOFTW_B : BOOL; (* wrong SW version operational msg. *)
	ucTJ_SOFTW : USINT; (* number of TJ with wrong SW version *)
	ucNumberOfCylinder : USINT; (* number of cylinders *)
	ZylZahl : USINT; (* number of cylinders for CAN-Comm. *)
	tTecError : ARRAY[0..4] OF _TecJetError; (* error status gas inject valves *)
	usTecErrCntMax : ARRAY[0..4] OF USINT; (* max value for wrong gas flow trans *)
	StopM : BOOL; (* TRUE=engine is stopped *)
	CANopen_error : UINT; (* CAN CONTROLLER STATUS 0=OK *)
	usTecErrCnt : ARRAY[0..4] OF USINT; (* counter for wrong gas flow transm. *)
	bSuctionMon : BOOL;
	bPump : BOOL; (* TRUE =  alarm turbo suction mon. *)
	ssTJ2_StzPkt : ARRAY[0..11] OF INT; (* scaling TecJet110 position *)
	ssTJ1_StzPkt : ARRAY[0..9] OF INT; (* scaling TecJet50 position *)
	ucSendParTJ : USINT; (* number of actual handled TecJet *)
	ucStateOfPar : USINT; (* state of parameter transmission *)
	bTecJetStatErr : BOOL; (* TRUE= problem status read *)
	bTecJetParErr : BOOL; (* TRUE= problem para. transmission *)
	ucParCount : USINT; (* counter for actual handled param. *)
	TON_SecondTick : TON; (* second tick TRUE for 0,1 sec. *)
	ucNextParTJ : USINT; (* number of actual  handled TecJet *)
	bTJ_CAN : ARRAY[0..4] OF BOOL; (* TJ CAN communication error *)
	TecJetVers : UINT; (* gas inject valve software version *)
	ucStatNr : USINT; (* read status value counter *)
	bTJ_SOFTW : BOOL; (* trigger for wrong SW version delay *)
	TON_SOFTW : TON; (* delay for wrong software version *)
	xSignScal_TJpos : xSignScal; (* scale TecJet valve opening *)
	TJ_CAN : BOOL; (* TJ CAN KOPPLUNG GESTÖRT *)
	TJ_SOFTW : BOOL := 0; (* TJ FALSCHE SOFTWARE *)
	TJ_GASD : BOOL := 0; (* TJ GASVORDRUCK NICHT ERFUELLT *)
	TJ_GAST : BOOL := 0; (* TJ GASTEMPERATUR NICHT ERFUELLT *)
	TJ_INT : BOOL := 0; (* TJ INTERNER FEHLER *)
	TJ_MECH : BOOL := 0; (* TJ MECHANISCHE FEHLFUNKTION *)
	TJ_MECH_B : BOOL; (* TJ mechanical error message *)
	ucTJ_MECH : USINT; (* valve with mechanic error *)
	TJ_CAN_B : BOOL; (* TJ CAN comm. error message *)
	ucTJ_CAN : USINT; (* vlave with CAN communication error *)
	TJ_GAST_B : BOOL; (* TJ gas temperature message *)
	ucTJ_GAST : USINT; (* valve with wrong gas temperature *)
	TJ_GASD_B : BOOL; (* TJ gas inlet pressure message *)
	ucTJ_GASD : USINT; (* valve with wrong inlet pressure *)
	TJ_INT_B : BOOL; (* TJ internal error message *)
	ucTJ_INT : USINT; (* valve with internal error *)
	TJ_GASN_B : BOOL; (* TJ gas flow not reached message *)
	ucTJ_GASN : USINT; (* valve with gas flow not reached *)
	AmmSeqCAN : AmmSequence; (* FUB can communication *)
	AmmSeqGASD : AmmSequence; (* FUB gas pressure*)
	AmmSeqGASM : AmmSequence; (* FUB gas flow change *)
	AmmSeqGASN : AmmSequence; (* FUB gas flow not reached *)
	AmmSeqGASO : AmmSequence; (* FUB gas flow max. reached *)
	AmmSeqGAST : AmmSequence; (* FUB wrong gas temperature *)
	AmmSeqINT : AmmSequence; (* FUB gas valve internal error *)
	AmmSeqMECH : AmmSequence; (* FUB gas valve malfunction *)
	TON_SecondTick_1 : TON;
	E_TEC : ARRAY[0..4] OF _tEventTEC; (* CAN events gas inject valve param. *)
	ssTJPos : ARRAY[0..4] OF INT; (* TecJet opening in permill *)
	TJ_GASN : BOOL := 0; (* TJ GASMENGE NICHT ERREICHT *)
	MM2VIS : MM2VIS_struct; (*Module VISU-Interface (Module --> VISU)*)
	ETecError : ARRAY[0..4] OF USINT;
	usWobbeAct : UINT;
	P : USINT;
	ulGasFlowN : ARRAY[0..4] OF UDINT;
	CANopen_CMS_GMU : CANopen;
	bNoInitDetected : BOOL := FALSE; (*allways true, except 1cycle on init up*)
	SIM_rGMU_Pr_DiffGas : ARRAY[0..4] OF REAL; (*Differential Pressure over device [mbar*10]*)
	SIM_rGMU_Pos_Valve_Rad : ARRAY[0..4] OF REAL; (*Valve Position [rad *10]*)
	SIM_rGMU_Pos_Valve_Prom : ARRAY[0..4] OF REAL; (*Valve Position [%o]*)
	SIM_rGMU_Pr_FuelGas : ARRAY[0..4] OF REAL; (*Fuel Gas Pressure at device inlet [mbar*10]*)
	SIM_rGMU_T_FuelGas : ARRAY[0..4] OF REAL; (*Fuel Gas Temperature at device inlet [°C *10]*)
	SIM_rGMU_Q_FuelGas : ARRAY[0..4] OF REAL; (*Fuel Gas Amount denormalized [l/s*1000]*)
	SIM_rGMU_D_FuelGas : ARRAY[0..4] OF REAL; (*Fuel Gas Density denormalized [kg/m3*1000]*)
	ulHWPNumTJ : ARRAY[0..4] OF UDINT; (* hardware part number gas inject valve *)
	ulSerNumTJ : ARRAY[0..4] OF UDINT; (* serial number gas inject valve *)
END_VAR
```

### Program Logical/GasMeteringUnit/GMU (IEC, version 4.11.0) - + Gas Flow and surge protection logic

- GMUCyclic.st (not readable text: treated as protected, skipped)

- GMUInit.st (not readable text: treated as protected, skipped)

#### GMU.var - Local variables
```iecst
(********************************************************************
 * COPYRIGHT -- INNIO Company
 ********************************************************************
 * Program: GMU
 * File: GMU.var
 * Author: WaldharM
 * Created: October 29, 2012
 ********************************************************************
 * Local variables of program GMU
 ********************************************************************)
VAR
	TON_Monitoring1 : TON;
	TON_Monitoring2 : TON;
	bMonitoring : ARRAY[0..4] OF BOOL;
	TJ_GasN : ARRAY[0..4] OF BOOL; (* TJ gas flow not reached error *)
	ucErrNr : USINT; (* counter error status value *)
	TJ_GasT : ARRAY[0..4] OF BOOL; (* TJ gas temperature error *)
	TJ_Int : ARRAY[0..4] OF BOOL; (* TJ internal error *)
	TJ_Mech : ARRAY[0..4] OF BOOL; (* TJ malfunction *)
	TJ_GasD : ARRAY[0..4] OF BOOL; (* TJ inlet pressure error *)
	xOpMode : OpMode;
	ucMeas : USINT; (* counter for TecJet meassure value *)
	tTecErrorOld : ARRAY[0..4] OF _TecJetError; (* last error status gas inject valve *)
	ucMonNr : USINT;
	ssGP_ZD : INT; (* gas inject valve pressure change *)
	ssGPold : ARRAY[0..4] OF INT; (* last gas inject valve pressure *)
	ssGrenz : INT; (* turbo suction monitoring limit *)
	xTOF_bLR_GasStop : TOF; (*load rejection function: gas stop active*)
	T_3096_OFF : TIME := T#7s; (*delay for 3096 re-activation*)
	b_3096_OFF_LR : BOOL := TRUE; (*enable switch off 3096 during load rejection*)
	tDelTime_GVOpen : TIME := T#7s;
	ucTecNr : USINT;
	bValS_GMU_Ok : ARRAY[0..4] OF BOOL; (* Overall status ok *)
	bMech_GMU_Err : ARRAY[0..4] OF BOOL; (* Valve malfunction *)
	bInt_GMU_Err : ARRAY[0..4] OF BOOL; (* Valve internal failure *)
	bFlow_GMU_SetErr : ARRAY[0..4] OF BOOL; (* flow demand failued *)
	bFlow_GMU_Min : ARRAY[0..4] OF BOOL; (* flow not reached *)
	bFlow_GMU_Down : ARRAY[0..4] OF BOOL; (* zero flow detected *)
	bPr_Diff_GMU_Down : ARRAY[0..4] OF BOOL; (* zero pressure detected *)
	bPos_GMU_Err : ARRAY[0..4] OF BOOL; (* Valve position failure *)
	bT_EU_GMU_HiHi : ARRAY[0..4] OF BOOL; (* Electronic temperature high *)
	bU_GMU_LoLo : ARRAY[0..4] OF BOOL; (* Input voltage low limit *)
	bT_GMU_LoLo : ARRAY[0..4] OF BOOL; (* 'Fuel gas temperature low limit *)
	bPr_Diff_GMU_LoLo : ARRAY[0..4] OF BOOL; (* Delta pressure low limit *)
	bPr_GMU_LoLo : ARRAY[0..4] OF BOOL; (* Fuel gas pressure low limit *)
	bU_GMU_HiHi : ARRAY[0..4] OF BOOL; (* Input voltage high limit *)
	bT_GMU_HiHi : ARRAY[0..4] OF BOOL; (* 'Fuel gas temperature high limit *)
	bPr_Diff_GMU_HiHi : ARRAY[0..4] OF BOOL; (* Delta pressure high limit *)
	bPr_GMU_HiHi : ARRAY[0..4] OF BOOL; (* Fuel gas pressure high limit *)
END_VAR
```

### Program Logical/GasMeteringUnit/tecjet (IEC, version 4.12.0) - + TecJet main

- tecjetCyclic.st (not readable text: treated as protected, skipped)

- tecjetInit.st (not readable text: treated as protected, skipped)

#### tecjet.var
```iecst
(*******************************************************************************
	tecjet : Type definitions for the tecjet

	This code is confidential and proprietary to the INNIO Company.
	It may not be used in any form, or reproduced in any manner, without the express
	written permission of the INNIO Company.
	Copyright, INNIO Company, 2019

	- calcualtion of different gas inject valve concerning parameters for gas sort 0
	- send parameter to gas inject valve
	- handling gas inject valve communication problem
	- read software version, operating hours, and gas inject valve status
	- check gas inject valve software version

	Customized modifications: -
	------------------------

	History:
	-------

	V3.99.0 07-04-2012  pankajrodey	,  Added new version for Modular software
	V3.99.1 27-11-2013  pankajrodey	,  Deleted variables to remove compilation warning

	Instructions for use:
	--------------------

	Outstandings:
	------------
	*******************************************************************************)
VAR
	TON_SendDelay : TON; (* FUB delay befor send Tecjet param. *)
	TJ_Softw : ARRAY[0..4] OF BOOL; (* TJ wrong software version *)
	AmmSeqTJ_SOFTW : AmmSequence; (* FUB AmmSeq. wrong SW version *)
	xTON_MeasVal : TON;
	ssGrenz : INT; (* turbo suction monitoring limit *)
	TJ_GasM : ARRAY[0..4] OF BOOL; (* TJ gas flow change error *)
	TJ_GasO : ARRAY[0..4] OF BOOL; (* TJ gas flow maximum error *)
	ucMeas : USINT; (* counter for TecJet meassure value *)
	ucTecNr : USINT;
END_VAR
```

- Logical/GasMeteringUnit/cmstec (protected, skipped)

### Program Logical/GasMeteringUnit/canmaiGD (IEC, version 4.00.0) - + CAN main for tecjet

- canmaiGDCyclic.st (not readable text: treated as protected, skipped)

### Program Logical/GasMeteringUnit/caninitGD (IEC, version 4.01.0) - + CAN init for tecjet

- caninitCyclic.st (not readable text: treated as protected, skipped)

### Program Logical/GasMeteringUnit/MsgGD (IEC, version 4.13.0) - + TecJet alarms

- MsgGDCyclic.st (not readable text: treated as protected, skipped)

- MsgGDInit.st (not readable text: treated as protected, skipped)

#### MsgGD.var
```iecst
(*******************************************************************************
	Msg_GMU : Alarms for the GMU module

	This code is confidential and proprietary to the INNIO Company.
	It may not be used in any form, or reproduced in any manner, without the express
	written permission of the INNIO Company.
	Copyright, INNIO Company, 2019

	- calcualtion of different gas inject valve concerning parameters for gas sort 0
	- send parameter to gas inject valve
	- handling gas inject valve communication problem
	- read software version, operating hours, and gas inject valve status
	- check gas inject valve software version

	Customized modifications: -
	------------------------

	History:
	-------

	V3.99.0 07-04-2012  pankajrodey	,  Added new version for Modular software

	Instructions for use:
	--------------------

	Outstandings:
	------------
	*******************************************************************************)
VAR
	bGnlTrip1_modlGMU : BOOL;
	bGnlTrip2_modlGMU : BOOL;
	bGnlTrip3_modlGMU : BOOL;
	bGnlWarning_modlGMU : BOOL;
	iAdrAmmBase2MM : UDINT;
	iAdrMM2AmmBase : UDINT;
	xMsg3093 : Msg;
	xMsg3094 : Msg;
	xMsg3095 : Msg;
	xMsg3096 : Msg;
	xMsg3098 : Msg;
	xMsg3097 : Msg;
	xMsg3213 : Msg;
	xMsg3241 : Msg;
	xMsg3242 : Msg;
	xMsg3243 : Msg;
	xMsg3244 : Msg;
	xMsg3245 : Msg;
	xMsg3246 : Msg;
	xMsg3249 : Msg;
END_VAR
```

### Program Logical/GasMeteringUnit/IN_GD (IEC, version 4.12.0) - + A new program

- IN_GDCyclic.st (not readable text: treated as protected, skipped)

### Program Logical/GasMeteringUnit/OUT_GD (IEC, version 4.05.0) - + OUT Task GasMeteringUnit

- OUT_GDCyclic.st (not readable text: treated as protected, skipped)

#### OUT_GD.var - Local variables
```iecst
(********************************************************************
 * COPYRIGHT -- INNIO Company
 ********************************************************************
 * Program: OUT_GMU
 * File: OUT_GMU.var
 * Author: 320003156
 * Created: February 17, 2012
 ********************************************************************
 * Local variables of program OUT_GMU
 ********************************************************************)
VAR
	I : USINT;
	iRev_HWP : ARRAY[0..4] OF UDINT;
	sRev_HWP : ARRAY[0..4] OF STRING[10];
	iNum_HWP : ARRAY[0..4] OF UDINT;
	sNum_HWP : ARRAY[0..4] OF STRING[10];
	sGMU_Num_HWP_tmp : ARRAY[0..4] OF STRING[10];
	sGMU_Num_HWP : ARRAY[0..4] OF STRING[10];
END_VAR
```

### can.var - Package variables
```iecst
VAR

	CMSTecJet_Init : CMSinit; (* FUB CAN CMS communication init *)

	CMSmain_TecJet : CMSmain; (* FUB for comm. to Tecjet *)

END_VAR
```

### Program Logical/GasMeteringUnit/VisGD (IEC, version 4.00.0) - + A new program

- VisGDCyclic.st (not readable text: treated as protected, skipped)

- VisGDInit.st (not readable text: treated as protected, skipped)

#### VisGD.var - Local variables
```iecst
(*******************************************************************************
	VisGMU : Update the VIS interfaces variable declaration

	This code is confidential and proprietary to the INNIO Company.
	It may not be used in any form, or reproduced in any manner, without the express
	written permission of the INNIO Company.
	Copyright, INNIO Company, 2019

	- calcualtion of different gas inject valve concerning parameters for gas sort 0
	- send parameter to gas inject valve
	- handling gas inject valve communication problem
	- read software version, operating hours, and gas inject valve status
	- check gas inject valve software version

	Customized modifications: -
	------------------------

	History:
	-------

	V3.99.1 28-08-2012  pankajrodey	,  Initial file

	Instructions for use:
	--------------------

	Outstandings:
	------------
	*******************************************************************************)

VAR
iIndex : INT;
END_VAR

VAR CONSTANT

END_VAR
```

### Program Logical/GasMeteringUnit/ParGD (IEC, version 4.06.0) - + Paramaters GasMeteringUnit

- perm_par.st (not readable text: treated as protected, skipped)

#### perm_par.var
```iecst
VAR
	tParaIntern : ParaHandler_typ; (*Connector type to perm_par*)
	tMM2ParaBase_ReadBack : MM2ParaBase_type; (*INTERNAL! V4.06 new readback structure for information from previous tasks*)
	bWriteDataObj : BOOL; (* TRUE=write data object module *)
	bDataObjLenErr : BOOL; (*Error occured in permem: data module size missmatch*)
	bCreateDataObj : BOOL; (* TRUE=create new data object *)
	bWriteOnce : BOOL; (* write permanent memory once *)
	DatObjCreate_01 : DatObjCreate; (* data object create *)
	DatObjInfoBak_02 : DatObjInfo; (* data object info *)
	DatObjDelete_01 : DatObjDelete; (* data object delete *)
	DatObjRead_01 : DatObjRead; (* data object read *)
	DatObjRead_02 : DatObjRead; (* manual initiated data object read *)
	DatObjWrite_01 : DatObjWrite; (* data object write *)
	DatObjDelete_02 : DatObjDelete; (* data object delete *)
	DatObjDelete_11 : DatObjDelete; (*Delete Backup File*)
	DatObjInfo_01 : DatObjInfo; (* data object info *)
	DatObjInfo_02 : DatObjInfo; (* data object info *)
	szModuleName : STRING[35]; (* module name of object *)
	szModuleNameBackup : STRING[35]; (* module name of posiibly created backup object *)
	DatObjCopy_01 : DatObjCopy;
	bCopyDataObj : BOOL;
	TON_WarnDelay : TON;
	TON_WritePMEM : TON; (* delay write permanent memory *)
	ulPMPointer : UDINT; (* adress of actual checksum value *)
	ulChecksum : UDINT; (* parameter checksum value *)
	pm_len : UDINT; (* permanent value lenght *)
	ulChecksumOld : UDINT; (* last vlaue of parameter checksum *)
	ulChkValue : UDINT; (* actual value of parameter pointer *)
	pm_id : UDINT; (* permanent value identifier *)
	pm_p : UDINT; (* permanent value pointer *)
	DatObjInfo_META : DatObjInfo;
	DatObjRead_META : DatObjRead;
	szMetaDataRaw : STRING[2000];
	szMetaData : ARRAY[0..4] OF STRING[35];
	szMetaDataVis : ARRAY[0..3] OF STRING[35];
	ssIndex : INT;
	ssCount : INT;
	ucMetaDataRaw : ARRAY[0..2000] OF USINT;
	ssCount2 : INT;
	szMetaDataFile : STRING[10];
	szText1 : STRING[20];
	pv_adr_IN_XX_tPB2MM : UDINT;
	pv_lng : UDINT;
	pv_lng_IN_XX_tPB2MM : UDINT;
	pv_lng_OUT_XX_tPB2MM : UDINT;
	szText2 : STRING[20];
	pv_adr_OUT_XX_tXX2PB : UDINT;
END_VAR
VAR CONSTANT
	ERR_NOERROR : UINT := 0;
END_VAR
VAR
	usPMWriteCnt : UINT;
	pm_Error : UDINT; (* permanent value error *) (* Deleted: pm : ParaMem_typ; permanent memory tags mathias, 22.8.11*)
	fun_Error : UDINT := 0; (*state > 0 = function error*)
	xLocalParaCheck : ParaCheckFUB; (*local function instance to check parameter values*)
	TON_ParaSetupOk : TON;
	bParaCheckSystemOk : BOOL;
	iDebug_ParaOkChecked : UDINT;
	bRestoreBackupDataObj : BOOL := FALSE;
	bRestoreDataObjContent : BOOL := FALSE;
	pm_id_backup : UDINT;
	pm_p_Backup : UDINT;
	DatObjCopy_02 : DatObjCopy;
	bDeleteBackupDataObj : BOOL := FALSE; (*Command to delete backup data module file on purpose*)
	bDebugPara : ARRAY[0..5] OF BOOL;
	ssIndex2 : INT;
	ssIndex3 : INT;
	ssIndex4 : INT;
	ssIndexVis : INT;
	szText : STRING[40];
	pv_adr_Para : UDINT;
	szParaSnippet : ARRAY[0..5] OF STRING[150];
	szParaIndex : STRING[10];
	slValue : DINT;
	iModuleDLD_ResetCount : INT;
	bDownloadDetected : BOOL;
	bFlagParaStructCopyWorking : BOOL; (*true, if cyclic para copying is active, 1 false cycle at every copy *)
	bStoreInitParaInDataObj : BOOL := FALSE;
	bTestflag : BOOL;
	bReadOutMETA_Once : BOOL;
	tParaCheck_iPvAdress : ARRAY[0..5] OF UDINT;
	tParaCheck_iPvLengt : ARRAY[0..5] OF UDINT;
	tParaCheck_rPvValue : ARRAY[0..5] OF REAL;
	tParaCheck_rRangeMIN : ARRAY[0..5] OF REAL;
	tParaCheck_rRangeMAX : ARRAY[0..5] OF REAL;
	tParaCheck_szPvName : ARRAY[0..5] OF STRING[35];
	ssFormatDetected : INT;
	szMetaDataPart : STRING[150];
	szFullTaskName : STRING[35];
	szFullMetaModuleName : STRING[35];
	debugLen : INT;
	debugSize : INT := 0;
	strcat_adr1 : UDINT;
	strcat_adr2 : UDINT;
	ssIndexTN : INT;
	bAlternate : BOOL;
	n : INT;
	iAlternateChecksum : DINT;
	iAlternateChecksumOld : DINT;
	ulDebugChkValue : ARRAY[0..999] OF UDINT;
	Adr1 : UDINT;
	Adr2 : UDINT;
	usPMWriteCntStepsize : UINT := 1; (*different step sizes to help debug*)
	usPMWriteCntXOR : UINT;
	usPMWriteCntAltSum : UINT;
	ulAdrPM : UDINT;
	usChkValuePM : USINT;
	ulAdrPara : UDINT;
	ulPara_len : UDINT;
	usChkValuePara : USINT;
	iDebugCountPMDifferences : DINT := 0;
	bEngineRunDetected : BOOL; (*detection status bit autocommand 100 /101  for engine run state*)
	ucMetaDataDebugInfoLine : ARRAY[0..24] OF STRING[80];
	ssIndexMand : INT := 0;
	szMetaDataMand : STRING[35];
	iMyErrorInfo_Autoreset : DINT; (*internal autoreset counter*)
	ssIndex_Version : INT; (*internal*)
	ssIndex_BU : INT; (*internal*)
	ssIndex_BU2 : INT; (*internal*)
END_VAR
```

### Package Logical/Gasmixer - GM: Gas Mixer

### Data object Logical/Gasmixer/META_GM (Simple) - MODUL META data file

#### META_GM.dat
```
; *******************************************************************************
; AGGR: Module Meta Data (data module)
;
; This code is confidential and proprietary to the INNIO Company.
; It may not be used in any form, or reproduced in any manner, without the express
; written permission of the INNIO Company.
; Copyright, INNIO Company, 2021
;
; Customized modifications: -
; ------------------------
;
; History:
; -------
; V03.99.00.00	06.03.2013	Weitzer 	generated for modular software
; V04.00.00.00	31.01.2014	Weitzer 	versions changed
; V04.01.00.00	14.06.2014	Weitzer 	special gasmixer added
; V04.05.00.00	22.01.2018	Tinello		Release Module added
; V04.05.01.00	20.02.2018	Tinello		Bugfix for measurement signal failure of gasmixer position
; V04.07.01.00	17.10.2019	Tinello		bugfix: division by 0
; V04.10.00.00	26.01.2021	Tinello		BugFix: Timer-FuB's
;
; Instructions for use:
; --------------------
; make only changes at the version numbers
;
; Outstandings:
; ------------
;
; *******************************************************************************
;
"<META>"
;
; Module ID
"<MODUL>GM</MODUL>"
;
; Module Version (xx.yy.zz.cc)
"<VERSION>04.10.00.00</VERSION>"
;
; Module Basisupdate Version BU (00-99)
"<BASISUPDATE_VERSION>00</BASISUPDATE_VERSION>"
;
; Optional: specify order number for limitated module usage
"<ORDER></ORDER>" ;<!--(optional for restricted customizations; missing statement makes module valid for all orders)-->
;
; Parameter Check <PARAn Name='aAbcdef' MIN='xxx' MAX='yyy' />  (watch for correct spacings and apostrophs!)
"<PARAMETER_CHK>"
"<PARA1 Name='iEng_Motortype' MIN='208' MAX='920' />"
"<PARA2 />"
"<PARA3 />"
"<PARA4 />"
"<PARA5 />"
"</PARAMETER_CHK>"
;
; Permanent Datamodule Filenames<!-- NAME ist ohne Dateiendung einzutragen; Nur für Counter und interne Parameter verwenden-->
"<DATAMODULES>" ;<!-- optional; mehrere DATAMODULES erlaubt-->
"	<DATAMODULE>par_GM</DATAMODULE>"
"</DATAMODULES>"
;
; Dependencies Modules (MMxx.yy.zz.cc)
"<DEPENDENCIES>"
"	<DEPENDENCY MODULE='AB' VERSION='04.00.00.00' />"
"	<DEPENDENCY MODULE='AG' VERSION='04.01.00.00' />"
"	<DEPENDENCY MODULE='PB' VERSION='04.00.00.00' />"
"	<DEPENDENCY MODULE='HA' VERSION='04.04.00.00' />"
"	<DEPENDENCY MODULE='OP' VERSION='04.01.00.00' />"
"	<DEPENDENCY MODULE='EC' VERSION='04.00.00.00' />"
"	<DEPENDENCY MODULE='GT' VERSION='04.00.00.00' />"
"	<DEPENDENCY MODULE='IG' VERSION='04.00.00.00' />"
"   <DEPENDENCY VISVERSION='02.01.00.00' />"			; Dependencies Visualization
"</DEPENDENCIES>"
;
; Module function description
"<MODULEFUNCTION>" ;<!-- short overview documentation of module function; add reference to detailed information, if available-->
"	<General>	"
"	Control up to 2 gasmixer positions "
"	</General>	"
""
"	<F1 Name='Parameter sending' LastModified='04.00.00.00'>"
"	Send parameters and operation values to the device.	"
"	</F1>"
"	<F2 Name='Referencing' LastModified='04.00.00.00'>"
"	Set reference position of stepper motor driver	"
"	</F2>"
"	<F3 Name='Monitor difference' LastModified='04.00.00.00'>"
"	Monitor difference between analog position and stepper position	"
"	</F3>"
"	<F4 Name='BugFix' LastModified='04.10.00.00'>"
"	BugFix: Timer-FuB's"
"	</F4>"
""
"	<Info>"
"	Please enter additional module info here.	"
"	</Info>"
""
"	<Customized LastModified='04.00.00.00'>	"
"	- Nothing "
"	</Customized>	"
""
"</MODULEFUNCTION>"
;
"</META>"
```

### Module_GasMixer.typ - Module global data types
```iecst
TYPE
	IN_GM_Struct : 	STRUCT
		bLeanox_Active : BOOL; (*leanox controller is active*) (*OldName: bLeanoxActive; Cycle: 5;*) (*V04.00.00.00*)
		bLeanox_Man : BOOL; (*leanox controller in manual*) (*OldName: l_einst_a; Cycle: 5;*) (*V04.00.00.00*)
		bSimWinMOD_Active : BOOL; (*WinMode simulation active*) (*OldName: new PV; Cycle: 5;*) (*V04.04.00.00*)
		iGM1_MStepActPos : DINT; (*gasmixer 1 - Actual position from SM1426-Module [Microsteps]*) (*OldName: slGM1_MStepActPos_TC1; Cycle: 5;*) (*V04.00.00.00*)
		iGM1_Status : UINT; (*gasmixer 1 - Status Word from SM1426-Module*) (*OldName: usGM1_Status_TC1; Cycle: 5;*) (*V04.00.00.00*)
		iGM2_MStepActPos : DINT; (*gasmixer 2 - Actual position from SM1426-Module [Microsteps]*) (*OldName: slGM2_MStepActPos_TC1; Cycle: 5;*) (*V04.00.00.00*)
		iGM2_Status : UINT; (*gasmixer 2 - Status Word from SM1426-Module*) (*OldName: usGM2_Status_TC1; Cycle: 5;*) (*V04.00.00.00*)
		iIdx_Gtyp_Dem : INT; (*actual gassort 1..4*) (*OldName: gasart; Cycle: 2;*) (*V04.00.02.00*)
		iIdx_OMSS : INT; (*operating mode selection switch (0=OFF/ 1=Hand/ 2=Auto/ 3=Test/ 4=Spülen)*) (*OldName: BWS_HA; Cycle: 5;*) (*V04.00.00.00*)
		iSt_OpMode : UDINT; (*engine operation mode*) (*OldName: StopM; Cycle: 5;*) (*V04.00.00.00*)
		rGT_QualMix_1_2 : REAL; (*Mixture ratio bet. gas 1 and 2 [%], e.g. value 0.75 = 75%*) (*OldName: ssMisch1_2; Cycle: 2;*) (*V04.00.02.00*)
		rN_EngAct : REAL; (*engine speed [rpm]*) (*OldName: n_ist; Cycle: 2;*) (*V04.00.02.00*)
		rP_Act_Norm_Filt : REAL; (*actual power related to rP_Nom filtered T=1s [%Pnom]*) (*OldName: P_IST; Cycle: 2;*) (*V04.00.02.00*)
		rP_Nom : REAL; (*nominal electric power, depends on gastype [kW]*) (*OldName: PN_GASART; Cycle: 2;*) (*V04.00.02.00*)
		rP_Set_Norm : REAL; (*power setpoint related to rP_Nom [%Pnom]*) (*OldName: p_soll; Cycle: 2;*) (*V04.00.02.00*)
		rPos_GM_Set_Norm : REAL; (*normed gasmixer set position [%]*) (*OldName: usStepperRatedPos; Cycle: 5;*) (*V04.00.00.00*)
		rPos_GM_Set_Norm_TC2 : REAL; (*normed gasmixer set position [%]*) (*OldName: usStepperRatedPos; Cycle: 2;*) (*V04.05.00.00*)
		tAB2GM : AmmBase2MM; (*AMM structure*) (*OldName: QUITTRPS; Cycle: 5;*) (*V04.00.00.00*)
		tPB2MM : ParaBase2MM_type; (*Para structure*) (*OldName: new PV; Cycle: 5;*) (*V04.00.00.00*)
		tPos_Act_GM1_Norm : HALioAi_Type; (*gasmixer 1 - normed actual position from potentiometer [%] (E.01-M-001)*) (*OldName: ssGasMixerPos1WE, AI_GasMixerPos1_TC1, ssGasMixerPos1; Cycle: 5;*) (*V04.00.00.00*)
		tPos_Act_GM2_Norm : HALioAi_Type; (*gasmixer 2 - normed actual position from potentiometer [%] (E.01-M-002)*) (*OldName: ssGasMixerPos2WE, AI_GasMixerPos2_TC1, ssGasMixerPos2; Cycle: 5;*) (*V04.00.00.00*)
		tPos_SGM_Enc1 : HALioAi_INT_Type; (*SGM encoder position stepper 1 [1]*) (*OldName: ss1EncPos_we; Cycle: 2;*) (*V04.00.02.00*)
		tPos_SGM_Enc2 : HALioAi_INT_Type; (*SGM encoder position stepper 1 [1]*) (*OldName: ss1EncPos_we; Cycle: 2;*) (*V04.00.02.00*)
		tPos_SGM_Enc3 : HALioAi_INT_Type; (*SGM encoder position stepper 1 [1]*) (*OldName: ss1EncPos_we; Cycle: 2;*) (*V04.00.02.00*)
	END_STRUCT;
	MM2VIS_Struct : 	STRUCT
		bMsg1083 : BOOL; (*Prio2: error gasmixer control*) (*OldName: M_RPSA11; Cycle: 5;*) (*V04.00.00.00*)
		bMsg2086 : BOOL; (*Prio4: measuring signal failure gasmixer position*) (*OldName: M_RPSW6; Cycle: 5;*) (*V04.00.00.00*)
		bSGM_RefActive : BOOL; (*SGM reference check is running*) (*OldName: M_GM_Ref; Cycle: 2;*) (*V04.00.02.00*)
		rPos_Act_GM1_Norm : REAL; (*gasmixer 1 - normed actual position [%]*) (*OldName: bp_y, ANA.LLPOS, ANA.TJ_y, S_K_W[137], S_K_W[142]; Cycle: 5;*) (*V04.00.00.00*)
		rPos_Act_GM2_Norm : REAL; (*gasmixer 2 - normed actual position [%]*) (*OldName: bp2_y; Cycle: 5;*) (*V04.00.00.00*)
		rPos_SGM_AirThrRel : REAL; (*SGM position air throttle in [mm]*) (*OldName: usLdrRel; Cycle: 2;*) (*V04.00.02.00*)
		rPos_SGM_GasThr : REAL; (*SGM position gas throttle in [%]*) (*OldName: usGasThrActPos; Cycle: 2;*) (*V04.00.02.00*)
		rPos_SGM_Stepper1 : REAL; (*SGM position encoder 1 [%]*) (*OldName: ss1EncPos; Cycle: 2;*) (*V04.00.02.00*)
		rPos_SGM_Stepper2 : REAL; (*SGM position encoder 2 [%]*) (*OldName: ss2EncPos; Cycle: 2;*) (*V04.00.02.00*)
		rPos_SGM_Stepper3 : REAL; (*SGM position encoder 3 [%]*) (*OldName: ss3EncPos; Cycle: 2;*) (*V04.00.02.00*)
	END_STRUCT;
	OUT_GM_Struct : 	STRUCT
		bEng_Bloc_SGM : BOOL; (*SGM blocks engine start because reference procedure is active *) (*OldName: M_GM_Ref; Cycle: 2;*) (*V04.00.02.00*)
		iGM1_Control : UINT; (*gasmixer 1 - Handover Control Word to SM1426-Module*) (*OldName: usGM1_Control_TC1; Cycle: 5;*) (*V04.00.00.00*)
		iGM1_Mode : SINT; (*gasmixer 1 - Handover Mode to SM1426-Module*) (*OldName: scGM1_Mode_TC1; Cycle: 5;*) (*V04.00.00.00*)
		iGM1_MStepSetPos : DINT; (*gasmixer 1 - Handover Set position to SM1426-Module [Microsteps]*) (*OldName: slGM1_MStepSetPos_TC1; Cycle: 5;*) (*V04.00.00.00*)
		iGM2_Control : UINT; (*gasmixer 2 - Handover Control Word to SM1426-Module*) (*OldName: usGM2_Control_TC1; Cycle: 5;*) (*V04.00.00.00*)
		iGM2_Mode : SINT; (*gasmixer 2 - Handover Mode to SM1426-Module*) (*OldName: scGM2_Mode_TC1; Cycle: 5;*) (*V04.00.00.00*)
		iGM2_MStepSetPos : DINT; (*gasmixer 2 - Handover Set position to SM1426-Module [Microsteps]*) (*OldName: slGM2_MStepSetPos_TC1; Cycle: 5;*) (*V04.00.00.00*)
		tGM2AB : MM2AmmBase; (*AMM structure*) (*OldName: new PV; Cycle: 5;*) (*V04.00.00.00*)
		tGM2PB : MM2ParaBase_type; (*Para structure*) (*OldName: new PV; Cycle: 5;*) (*V04.00.00.00*)
		tSGM_DirStepper1 : HALioDo_Type; (*DO SGM direction stepper 1*) (*OldName: b1StepperDir; Cycle: 2;*) (*V04.00.02.00*)
		tSGM_DirStepper2 : HALioDo_Type; (*DO SGM direction stepper 2*) (*OldName: b2StepperDir; Cycle: 2;*) (*V04.00.02.00*)
		tSGM_DirStepper3 : HALioDo_Type; (*DO SGM direction stepper 3*) (*OldName: b3StepperDir; Cycle: 2;*) (*V04.00.02.00*)
		tSGM_EnabStepper1 : HALioDo_Type; (*DO SGM enable stepper 1*) (*OldName: b1StepperEnab; Cycle: 2;*) (*V04.00.02.00*)
		tSGM_EnabStepper2 : HALioDo_Type; (*DO SGM enable stepper 2*) (*OldName: b2StepperEnab; Cycle: 2;*) (*V04.00.02.00*)
		tSGM_EnabStepper3 : HALioDo_Type; (*DO SGM enable stepper 3*) (*OldName: b3StepperEnab; Cycle: 2;*) (*V04.00.02.00*)
	END_STRUCT;
	PARA_GM_Struct : 	STRUCT
		bLeanox_Speed_Exist : BOOL; (*PARA [11060]: TRUE = leanox in island mode active*) (*OldName: lox_np_akt; Cycle: 2;*) (*V04.00.02.00*)
		bSGM_Active : BOOL; (*PARA [12362]: Special Gas Mixer (SGM) active*) (*OldName: bSpecGM; Cycle: 2;*) (*V04.00.02.00*)
		iEng_Motortype : INT; (*PARA [00000]: engine motortype*) (*OldName: motortyp; Cycle: 5;*) (*V04.00.00.00*)
		iF_SGM_Stepper1 : UINT; (*PARA [12382]: SGM stepper 1 speed of steps [Hz]*) (*OldName: sgm_lox_speed1; Cycle: 2;*) (*V04.00.02.00*)
		iF_SGM_Stepper2 : UINT; (*PARA [12383]: SGM stepper 2 speed of steps [Hz]*) (*OldName: sgm_lox_speed2; Cycle: 2;*) (*V04.00.02.00*)
		iF_SGM_Stepper3 : UINT; (*PARA [12384]: SGM stepper 3 speed of steps [Hz]*) (*OldName: sgm_lox_speed3; Cycle: 2;*) (*V04.00.02.00*)
		iNum_GM : INT; (*PARA [11357]: number of gasmixer*) (*OldName: AnzGasm; Cycle: 5;*) (*V04.00.00.00*)
		iNum_SGM_FullStepStepper1 : UINT; (*PARA [12379]: SGM stepper 1 number of full steps [1]*) (*OldName: sgm_full_step1; Cycle: 2;*) (*V04.00.02.00*)
		iNum_SGM_FullStepStepper2 : UINT; (*PARA [12380]: SGM stepper 2 number of full steps [1]*) (*OldName: sgm_full_step2; Cycle: 2;*) (*V04.00.02.00*)
		iNum_SGM_FullStepStepper3 : UINT; (*PARA [12381]: SGM stepper 3 number of full steps [1]*) (*OldName: sgm_full_step3; Cycle: 2;*) (*V04.00.02.00*)
		rNum_stepsGM1 : REAL; (*PARA [11358]: number of half-steps for 100% gasmixer 1 opening*) (*OldName: full_step; Cycle: 5;*) (*V04.00.00.00*)
		rNum_stepsGM2 : REAL; (*PARA [11359]: number of half-steps for 100% gasmixer 2 opening*) (*OldName: full_step1; Cycle: 5;*) (*V04.00.00.00*)
		rP_Leanox_Act_SP : ARRAY[0..4]OF REAL; (*PARA [11163]: Leanox activation switching point [kW]*) (*OldName: lox_st; Cycle: 2;*) (*V04.00.02.00*)
		rPos_SGM_AirThrFullLoad : ARRAY[0..4]OF REAL; (*PARA [12363]: SGM position gas throttle at full laod [mm]*) (*OldName: LdrVoll; Cycle: 2;*) (*V04.00.02.00*)
		rPos_SGM_AirThrOffsIdle : ARRAY[0..4]OF REAL; (*PARA [12367]: SGM offset air throttle at idle mode [mm]*) (*OldName: OfLdrLl; Cycle: 2;*) (*V04.00.02.00*)
		rPos_SGM_AirThrOffsNetp : ARRAY[0..4]OF REAL; (*PARA [12371]: SGM offset air throttle at net para mode [mm]*) (*OldName: OfLdrNp; Cycle: 2;*) (*V04.00.02.00*)
		rPos_SGM_AirThrOffsStart : ARRAY[0..4]OF REAL; (*PARA [12375]: SGM offset air throttle at engine start [mm]*) (*OldName: OfLdrSt; Cycle: 2;*) (*V04.00.02.00*)
	END_STRUCT;
	VIS2MM_Struct : 	STRUCT
		bSGM_Init : BOOL; (*start SGM reference check*) (*OldName: bInitSGM; Cycle: 2;*) (*V04.00.02.00*)
		bSGM_Man : BOOL; (*switch SGM to manual mode*) (*OldName: bGM_Man; Cycle: 2;*) (*V04.00.02.00*)
		rPos_SGM_SetStepper1 : REAL; (*SGM rated stepper position 1 [%]*) (*OldName: ss1StepRat; Cycle: 2;*) (*V04.00.02.00*)
		rPos_SGM_SetStepper2 : REAL; (*SGM rated stepper position 2 [%]*) (*OldName: ss2StepRat; Cycle: 2;*) (*V04.00.02.00*)
		rPos_SGM_SetStepper3 : REAL; (*SGM rated stepper position 3 [%]*) (*OldName: ss3StepRat; Cycle: 2;*) (*V04.00.02.00*)
	END_STRUCT;
END_TYPE
```

### Module_GasMixer.var - Module global variables
```iecst
VAR
	bErrGM_Ctr : BOOL := FALSE; (*Error gasmixer control*)
	bErrMsGM_Pos : BOOL := FALSE; (*Error measurement signal -  gasmixer position*)
	bErrSGM_Ctr : BOOL; (*Error special gas mixer*)
	bGnlTrip : BOOL; (*general alarm trip *)
	bGnlTrip1 : BOOL; (*general alarm trip priority 1*)
	bGnlTrip2 : BOOL; (*general alarm trip priority 2*)
	bGnlTrip3 : BOOL; (*general alarm trip priority 3*)
	bGnlWarning : BOOL; (*general alarm warning *)
	bNoInitDetected : BOOL := FALSE; (*allways true, except 1cycle on init up*)
	bOMSS_MAT : BOOL; (*operation mode selector switch - MANUAL/AUTO/TEST*)
	bRelModul_ParaSetupOk : BOOL := FALSE; (*Release Module if ParaSetupOk = TRUE*) (* *) (*V04.05.00.00*)
	IN_GM : IN_GM_Struct; (*Module IN-Interface*)
	MM2VIS : MM2VIS_Struct; (*Module VISU-Interface (Module --> VISU)*)
	OUT_GM : OUT_GM_Struct; (*Module OUT-Interface*)
	Para : PARA_GM_Struct; (*Module Parameter-Interface*)
	ParaFactoryDefault : PARA_GM_Struct := (0); (*First Init Values*)
	pm : PARA_GM_Struct; (*Stored parameter structure *)
	VIS2MM : VIS2MM_Struct; (*Module VISU-Interface (VISU --> Module)*)
	xOpMode : OpMode := (0); (*FuB*)
END_VAR
```

### Program Logical/Gasmixer/GeneralGM (IEC, version 4.00.0) - general functions

#### GeneralGMCyclic.st - Cyclic code
```iecst
(*******************************************************************************
GeneralGM		general functions

This code is confidential and proprietary to the INNIO Company.
It may not be used in any form, or reproduced in any manner,
without the express written permission of the INNIO Company.
Copyright, INNIO Company, 2019

Customized modifications: -
------------------------

History:
-------
V03.99.00.00	23.01.2013 	Tinello 	Created initial structured text code
V04.05.00.00	22.01.2018	Tinello		Release Module added

(*******************************************************************************)

PROGRAM _CYCLIC

	(* Release Module if ParaSetupOk = TRUE *)
	xTON_ParaSetupOk(IN		:= IN_GM.tPB2MM.bParaSetupOk, PT:= T#20s);
	bRelModul_ParaSetupOk	:= xTON_ParaSetupOk.Q;

	(* Operation mode selector switch *)
	bOMSS_MAT := (IN_GM.iIdx_OMSS = 1) OR (IN_GM.iIdx_OMSS = 2) OR (IN_GM.iIdx_OMSS = 3); (* 1= manual; 2= auto; 3= test mode *)

	(* call function for the state machine - engine operation mode *)
	xOpMode(in 	:= IN_GM.iSt_OpMode);

END_PROGRAM
```

#### GeneralGM.var - Local variables
```iecst
VAR
	xTON_ParaSetupOk : TON := (0); (*FuB*)
END_VAR
```

### Program Logical/Gasmixer/GM_control (IEC, version 4.10.0) - Gasmixer control

#### GM_controlCyclic.st - Cyclic code
```iecst
(************************************************************************************************************************************
GasMixer: control up to 2 gasmixer positions  (cyclic)

This code is confidential and proprietary to the INNIO Company.
It may not be used in any form, or reproduced in any manner,
without the express written permission of the INNIO Company.
Copyright, INNIO Company, 2021

	- convert analog gasmixer position to 1/100 %
	- check gasmixer position measurement signal
	- monitor difference between analog position and stepper position
	- set reference position of stepper motor driver

Customized modifications: -
------------------------

History:
-------
V03.99.00.00	07.01.2009	Tinello		generated from gasmixer-task V0.32
				19.02.2010	WeitzerT	replace QUITT_WA / _AB by QUITTRPS/ (QUITTRPS AND StopM)
				17.03.2010	WeitzerT	re-config and re-para if module was disconnected
				13.07.2011	lettenb.	line 328 slGM2_MStepSetPos_TC1: bp_y -> bp2_y bugfix for second SM1426
				10.01.2013	Tinello		restructured for Modulare SW
V04.01.00.00	13.06.2014	Weitzer		add bit for special gasmixer trip 1083
V04.04.00.00	21.12.2016	Denk		Modification for WinMOD simulation
V04.05.01.00	20.02.2018	Tinello		Bugfix for measurement signal failure of gasmixer position
V04.07.01.00	17.10.2019	Tinello		bugfix: division by 0
V04.10.00.00	27.01.2021	Tinello  	BugFix: Timer-FuB's

Instructions for use: -
--------------------

Outstandings: -
------------

*************************************************************************************************************************************)
PROGRAM _CYCLIC

	xTON_Referencing(IN := NOT xTON_Referencing.Q, PT:= T#9s980ms);				(* timer tick  10 s = 9980ms + 2 task class cycles	*)

	(*--------------------------------------------------*)
	(* RESET of alarms and warnings 					*)
	(*--------------------------------------------------*)
	bErrMsGM_Pos 	:= FALSE;
	bErrGM_Ctr		:= FALSE;

	(*--------------------------------------------------*)
	(* VISU var of module 								*)
	(*--------------------------------------------------*)
	MM2VIS.rPos_Act_GM1_Norm;
	MM2VIS.rPos_Act_GM2_Norm;

	(********************************************************************************************************************************)
	(* 													gasmixer 1 																	*)
	(********************************************************************************************************************************)
	IF Para.iNum_GM >= 1 AND IN_GM.tPB2MM.bParaSetupOk AND NOT Para.bSGM_Active AND NOT IN_GM.bSimWinMOD_Active THEN

		(*----------------------------------------------*)
		(* READ status from state machine				*)
		(*----------------------------------------------*)
		xWDtoBIT_GM1.Word 		:= IN_GM.iGM1_Status;
		xWDtoBIT_GM1();

		bGM1_ReadyToSwitchOn	:= xWDtoBIT_GM1.Bit00;
		bGM1_SwitchedOn			:= xWDtoBIT_GM1.Bit01;
		bGM1_OperationEnable	:= xWDtoBIT_GM1.Bit02;							(* ONLY state where motor movements are executed	*)
		bGM1_Error				:= xWDtoBIT_GM1.Bit03;
		bGM1_SwitchOnDisabled	:= xWDtoBIT_GM1.Bit06;
		bGM1_Warning			:= xWDtoBIT_GM1.Bit07;
		bGM1_TargetReached		:= xWDtoBIT_GM1.Bit10;							(* gets TRUE when an activity is finished 			*)

		(*----------------------------------------------*)
		(* CHANGE STATE 								*)
		(*----------------------------------------------*)
		IF    bGM1_SwitchedOn 		THEN 	bGM1_EnableVoltage		:= TRUE;	(* COMMAND: change state to "Operation Enable"		*)
											bGM1_SwitchOn			:= TRUE;
											bGM1_EnableOperation	:= TRUE;
		ELSIF bGM1_ReadyToSwitchOn 	THEN 	bGM1_EnableVoltage		:= TRUE;	(* COMMAND: change state to "Switched On"			*)
											bGM1_SwitchOn			:= TRUE;
											bGM1_EnableOperation	:= FALSE;
		ELSIF bGM1_SwitchOnDisabled THEN 	bGM1_EnableVoltage		:= TRUE;	(* COMMAND: change state to "Ready To Switch On"	*)
											bGM1_SwitchOn			:= FALSE;
											bGM1_EnableOperation	:= FALSE;	END_IF

		(* Acknowledgement *)
		IF IN_GM.tAB2GM.bResetWarning 				   AND bGM1_Warning	THEN  bGM1_ResetWarning	:= TRUE;	END_IF
		IF IN_GM.tAB2GM.bResetWarning AND xOpMode.Stop AND bGM1_Error	THEN  bGM1_ResetError	:= TRUE; 	END_IF

		(*----------------------------------------------*)
		(* WRITE COMMAND to state machine 				*)
		(*----------------------------------------------*)
		xBITtoWD_GM1.Bit00	:= bGM1_SwitchOn;
		xBITtoWD_GM1.Bit01	:= bGM1_EnableVoltage;
		xBITtoWD_GM1.Bit02	:= TRUE;
		xBITtoWD_GM1.Bit03	:= bGM1_EnableOperation;
		xBITtoWD_GM1.Bit07	:= bGM1_ResetError;									(* rising Edge to reset *)
		xBITtoWD_GM1.Bit12	:= bGM1_ResetWarning;								(* rising Edge to reset *)
		xBITtoWD_GM1();

		OUT_GM.iGM1_Control	:= xBITtoWD_GM1.Word;

		(* Reset Acknowledgement	*)
		bGM1_ResetError		:= FALSE;
		bGM1_ResetWarning	:= FALSE;

		(*----------------------------------------------*)
		(* CONVERT actual position from SM1426  		*)
		(*----------------------------------------------*)
		(* traversing range (Verfahrbereich) *)
		rGM1_MStepRange			:= Para.rNum_stepsGM1 / 2 * 256;			(* conversion from half-step to full-step to Microstep	*)

		IF rGM1_MStepRange <> 0 THEN
			rPos_Act_GM1_Norm	:= DINT_TO_REAL(IN_GM.iGM1_MStepActPos) / rGM1_MStepRange;	(* normed gasmixer position from SM1426	*)
		END_IF

		(*----------------------------------------------*)
		(* ERROR 										*)
		(*----------------------------------------------*)
		(* difference between potentiometer and SM1426 position > 1% for longer than 30 seconds or State Machine = "Fault" *)
		xTON_GM1_Err(IN := ABS(rPos_Act_GM1_Norm - IN_GM.tPos_Act_GM1_Norm.Unfilt) > 0.01, PT:= T#30s);
		bErrGM_Ctr 		:= xTON_GM1_Err.Q OR bGM1_Error;																(* A1083 *)

		(* measurement signal failure 	*)
		bErrMsGM_Pos	:= NOT IN_GM.tPos_Act_GM1_Norm.GoodQual;														(* W2086 *)

		(*----------------------------------------------*)
		(* SET position									*)
		(*----------------------------------------------*)
		IF 	bGM1_OperationEnable AND 				(* STATE Machine: motor movements are executed *)
			OUT_GM.iGM1_Mode = 1 					(* Position MODE: move to target position if actual position <> set position	*)
		THEN
			OUT_GM.iGM1_MStepSetPos	:= REAL_TO_DINT( rGM1_MStepRange * IN_GM.rPos_GM_Set_Norm);
		END_IF

		(*----------------------------------------------*)
		(* REFERENCING 									*)
		(*----------------------------------------------*)

		(* Calculate position error *)
		rPos_GM1_SumError_Norm	:= rPos_GM1_SumError_Norm + (rPos_Act_GM1_Norm - IN_GM.tPos_Act_GM1_Norm.Unfilt);
		rCnt_GM1_SumError		:= rCnt_GM1_SumError + 1;

		(* Set reference if acknowledge *)
		IF IN_GM.tAB2GM.bResetWarning AND xOpMode.Stop 	THEN  bGM1_SetRef	:= TRUE; 	END_IF

		IF (NOT IN_GM.bLeanox_Man OR 										(* leanox control not manual  	*)
			NOT xOpMode.Stop 	  OR 										(* engine is running 			*)
			bGM1_SetRef			 	) AND 									(* COMMAND: Set reference 		*)
			bGM1_OperationEnable 											(* STATE Machine: Set of actual position is allowed *)
		THEN

			IF 	xTON_Referencing.Q THEN										(* release referencing every 10s	*)

				(* Calculate normed average position error *)
				rPos_GM1_AvgError_Norm		:= rPos_GM1_SumError_Norm / rCnt_GM1_SumError;
				rPos_GM1_SumError_Norm		:= 0;
				rCnt_GM1_SumError			:= 0;

				(* if positioning error is > 0.2% and < 1.0% or engine stop and error is > 0.1% carry out a reference set *)
				IF 	(ABS(rPos_GM1_AvgError_Norm) > 0.002 AND ABS(rPos_GM1_AvgError_Norm) < 0.01) OR
					(xOpMode.Stop AND ABS(rPos_GM1_AvgError_Norm) > 0.001)
				THEN
					OUT_GM.iGM1_MStepSetPos := IN_GM.iGM1_MStepActPos - (REAL_TO_DINT(rGM1_MStepRange * rPos_GM1_AvgError_Norm) / 2);
					OUT_GM.iGM1_Mode	  	:= -122;						(* MODE: Set actual position  *)
				END_IF

				(* carry out a reference set *)
				IF bGM1_SetRef AND OUT_GM.iGM1_Mode <> -122
				THEN
					OUT_GM.iGM1_MStepSetPos	:= REAL_TO_DINT(rGM1_MStepRange * IN_GM.tPos_Act_GM1_Norm.Ai);
					OUT_GM.iGM1_Mode		:= -122;						(* MODE: Set actual position  *)
				END_IF

			ELSIF bGM1_TargetReached AND OUT_GM.iGM1_Mode = -122
			THEN
				OUT_GM.iGM1_Mode	:= 1;									(* Position MODE: Release for Set positioning	*)
				bGM1_SetRef			:= FALSE;								(* Reset COMMAND: Set reference *)
			END_IF
		END_IF

		(*----------------------------------------------*)
		(* VISU: normed gasmixer position  				*)
		(*----------------------------------------------*)
		IF NOT xOpMode.Stop THEN											(* if engine is running	*)
  			MM2VIS.rPos_Act_GM1_Norm	:= rPos_Act_GM1_Norm;				(* normed gasmixer position from SM1426 module *)
		ELSE
			MM2VIS.rPos_Act_GM1_Norm	:= IN_GM.tPos_Act_GM1_Norm.Ai;		(* filtered and normed gasmixer pos. from potentiometer *)
		END_IF

	ELSE
		OUT_GM.iGM1_Mode	:= 0;											(* NO MODE	*)
		bGM1_SetRef			:= TRUE;										(* carry out a reference set *)
		xTON_GM1_Err(IN 	:= FALSE);
	END_IF

	(********************************************************************************************************************************)
	(* 													gasmixer 2 																	*)
	(********************************************************************************************************************************)
	IF Para.iNum_GM >= 2 AND IN_GM.tPB2MM.bParaSetupOk AND NOT Para.bSGM_Active AND NOT IN_GM.bSimWinMOD_Active THEN

		(*----------------------------------------------*)
		(* READ status from state machine				*)
		(*----------------------------------------------*)
		xWDtoBIT_GM2.Word 		:= IN_GM.iGM2_Status;
		xWDtoBIT_GM2();

		bGM2_ReadyToSwitchOn	:= xWDtoBIT_GM2.Bit00;
		bGM2_SwitchedOn			:= xWDtoBIT_GM2.Bit01;
		bGM2_OperationEnable	:= xWDtoBIT_GM2.Bit02;							(* ONLY state where motor movements are executed	*)
		bGM2_Error				:= xWDtoBIT_GM2.Bit03;
		bGM2_SwitchOnDisabled	:= xWDtoBIT_GM2.Bit06;
		bGM2_Warning			:= xWDtoBIT_GM2.Bit07;
		bGM2_TargetReached		:= xWDtoBIT_GM2.Bit10;							(* gets TRUE when an activity is finished 			*)

		(*----------------------------------------------*)
		(* CHANGE STATE 								*)
		(*----------------------------------------------*)
		IF    bGM2_SwitchedOn 		THEN 	bGM2_EnableVoltage		:= TRUE;	(* COMMAND: change state to "Operation Enable"		*)
											bGM2_SwitchOn			:= TRUE;
											bGM2_EnableOperation	:= TRUE;
		ELSIF bGM2_ReadyToSwitchOn 	THEN 	bGM2_EnableVoltage		:= TRUE;	(* COMMAND: change state to "Switched On"			*)
											bGM2_SwitchOn			:= TRUE;
											bGM2_EnableOperation	:= FALSE;
		ELSIF bGM2_SwitchOnDisabled THEN 	bGM2_EnableVoltage		:= TRUE;	(* COMMAND: change state to "Ready To Switch On"	*)
											bGM2_SwitchOn			:= FALSE;
											bGM2_EnableOperation	:= FALSE;	END_IF

		(* Acknowledgement *)
		IF IN_GM.tAB2GM.bResetWarning 				   AND bGM2_Warning	THEN  bGM2_ResetWarning	:= TRUE;	END_IF
		IF IN_GM.tAB2GM.bResetWarning AND xOpMode.Stop AND bGM2_Error	THEN  bGM2_ResetError	:= TRUE; 	END_IF

		(*----------------------------------------------*)
		(* WRITE COMMAND to state machine 				*)
		(*----------------------------------------------*)
		xBITtoWD_GM2.Bit00	:= bGM2_SwitchOn;
		xBITtoWD_GM2.Bit01	:= bGM2_EnableVoltage;
		xBITtoWD_GM2.Bit02	:= TRUE;
		xBITtoWD_GM2.Bit03	:= bGM2_EnableOperation;
		xBITtoWD_GM2.Bit07	:= bGM2_ResetError;									(* rising Edge to reset *)
		xBITtoWD_GM2.Bit12	:= bGM2_ResetWarning;								(* rising Edge to reset *)
		xBITtoWD_GM2();

		OUT_GM.iGM2_Control	:= xBITtoWD_GM2.Word;

		(* Reset Acknowledgement	*)
		bGM2_ResetError		:= FALSE;
		bGM2_ResetWarning	:= FALSE;

		(*----------------------------------------------*)
		(* CONVERT actual position from SM1426  		*)
		(*----------------------------------------------*)
		(* traversing range (Verfahrbereich) *)
		rGM2_MStepRange			:= Para.rNum_stepsGM2 / 2 * 256;			(* conversion from half-step to full-step to Microstep	*)

		IF rGM2_MStepRange <> 0 THEN
			rPos_Act_GM2_Norm	:= DINT_TO_REAL(IN_GM.iGM2_MStepActPos) / rGM2_MStepRange;	(* normed gasmixer position from SM1426	*)
		END_IF

		(*----------------------------------------------*)
		(* ERROR 										*)
		(*----------------------------------------------*)
		(* difference between potentiometer and SM1426 position > 1% for longer than 30 seconds or State Machine = "Fault" *)
		xTON_GM2_Err(IN := ABS(rPos_Act_GM2_Norm - IN_GM.tPos_Act_GM2_Norm.Unfilt) > 0.01, PT:= T#30s);
		bErrGM_Ctr 		:= xTON_GM2_Err.Q OR bGM2_Error;																(* A1083 *)

		(* measurement signal failure 	*)
		bErrMsGM_Pos	:= bErrMsGM_Pos OR NOT IN_GM.tPos_Act_GM2_Norm.GoodQual;										(* W2086 *)

		(*----------------------------------------------*)
		(* SET position									*)
		(*----------------------------------------------*)
		IF 	bGM2_OperationEnable AND 				(* STATE Machine: motor movements are executed *)
			OUT_GM.iGM2_Mode = 1 					(* Position MODE: move to target position if actual position <> set position	*)
		THEN
			OUT_GM.iGM2_MStepSetPos	:= REAL_TO_DINT( rGM2_MStepRange * IN_GM.rPos_GM_Set_Norm);
		END_IF

		(*----------------------------------------------*)
		(* REFERENCING 									*)
		(*----------------------------------------------*)

		(* Calculate position error *)
		rPos_GM2_SumError_Norm	:= rPos_GM2_SumError_Norm + (rPos_Act_GM2_Norm - IN_GM.tPos_Act_GM2_Norm.Unfilt);
		rCnt_GM2_SumError		:= rCnt_GM2_SumError + 1;

		(* Set reference if acknowledge *)
		IF IN_GM.tAB2GM.bResetWarning AND xOpMode.Stop 	THEN  bGM2_SetRef	:= TRUE; 	END_IF

		IF (NOT IN_GM.bLeanox_Man OR 										(* leanox control not manual  	*)
			NOT xOpMode.Stop 	  OR 										(* engine is running 			*)
			bGM2_SetRef			 	) AND 									(* COMMAND: Set reference 		*)
			bGM2_OperationEnable 											(* STATE Machine: Set of actual position is allowed *)
		THEN

			IF 	xTON_Referencing.Q THEN										(* release referencing every 10s *)

				(* Calculate normed average position error *)
				rPos_GM2_AvgError_Norm		:= rPos_GM2_SumError_Norm / rCnt_GM2_SumError;
				rPos_GM2_SumError_Norm		:= 0;
				rCnt_GM2_SumError			:= 0;

				(* if positioning error is > 0.2% and < 1.0% or engine stop and error is > 0.1% carry out a reference set *)
				IF 	(ABS(rPos_GM2_AvgError_Norm) > 0.002 AND ABS(rPos_GM2_AvgError_Norm) < 0.01) OR
					(xOpMode.Stop AND ABS(rPos_GM2_AvgError_Norm) > 0.001)
				THEN
					OUT_GM.iGM2_MStepSetPos := IN_GM.iGM2_MStepActPos - (REAL_TO_DINT(rGM2_MStepRange * rPos_GM2_AvgError_Norm) / 2);
					OUT_GM.iGM2_Mode	  	:= -122;						(* MODE: Set actual position  *)
				END_IF

				(* carry out a reference set *)
				IF bGM2_SetRef AND OUT_GM.iGM2_Mode <> -122
				THEN
					OUT_GM.iGM2_MStepSetPos	:= REAL_TO_DINT(rGM2_MStepRange * IN_GM.tPos_Act_GM2_Norm.Ai);
					OUT_GM.iGM2_Mode		:= -122;						(* MODE: Set actual position  *)
				END_IF

			ELSIF bGM2_TargetReached AND OUT_GM.iGM2_Mode = -122
			THEN
				OUT_GM.iGM2_Mode	:= 1;									(* Position MODE: Release for Set positioning	*)
				bGM2_SetRef			:= FALSE;								(* Reset COMMAND: Set reference *)
			END_IF
		END_IF

		(*----------------------------------------------*)
		(* VISU: normed gasmixer position  				*)
		(*----------------------------------------------*)
		IF NOT xOpMode.Stop THEN											(* if engine is running	*)
  			MM2VIS.rPos_Act_GM2_Norm	:= rPos_Act_GM2_Norm;				(* normed gasmixer position from SM1426 module *)
		ELSE
			MM2VIS.rPos_Act_GM2_Norm	:= IN_GM.tPos_Act_GM2_Norm.Ai;		(* filtered and normed gasmixer pos. from potentiometer *)
		END_IF

	ELSE
		OUT_GM.iGM2_Mode	:= 0;											(* NO MODE	*)
		bGM2_SetRef			:= TRUE;										(* carry out a reference set *)
		xTON_GM2_Err(IN 	:= FALSE);
	END_IF

END_PROGRAM
```

#### GM_controlInit.st - Initialization code
```iecst
(*******************************************************************************
GasMixer: control up to 2 gasmixer positions  (init)

This code is confidential and proprietary to the INNIO Company.
It may not be used in any form, or reproduced in any manner,
without the express written permission of the INNIO Company.
Copyright, INNIO Company, 2019

Customized modifications: -
------------------------

History:
-------
V03.99.00.00	10.01.2013 	Tinello 	restructured

Instructions for use: -
--------------------

Outstandings: -
------------

(*******************************************************************************)
PROGRAM _INIT

	(* carry out a reference set *)
	bGM1_SetRef	:= TRUE;
	bGM2_SetRef	:= TRUE;

END_PROGRAM
```

#### GM_control.var - Local variables
```iecst
VAR
	bGM1_EnableOperation : BOOL := FALSE; (*gasmixer 1 - enable operation*)
	bGM1_EnableVoltage : BOOL := FALSE; (*gasmixer 1 - enable voltage*)
	bGM1_Error : BOOL := FALSE; (*gasmixer 1 - STATE: Error*)
	bGM1_OperationEnable : BOOL := FALSE; (*gasmixer 1 - STATE: operation enable*)
	bGM1_ReadyToSwitchOn : BOOL := FALSE; (*gasmixer 1 - STATE: ready to switch on*)
	bGM1_ResetError : BOOL := FALSE; (*gasmixer 1 - Reset Error*)
	bGM1_ResetWarning : BOOL := FALSE; (*gasmixer 1 - Reset Warning*)
	bGM1_SetRef : BOOL := TRUE; (*gasmixer 1 - COMMAND: Set Reference*)
	bGM1_SwitchedOn : BOOL := FALSE; (*gasmixer 1 - STATE: switched on*)
	bGM1_SwitchOn : BOOL := FALSE; (*gasmixer 1 - switch on*)
	bGM1_SwitchOnDisabled : BOOL := TRUE; (*gasmixer 1 - STATE: switch on disabled*)
	bGM1_TargetReached : BOOL := FALSE; (*gasmixer 1 - STATE: targed reached*)
	bGM1_Warning : BOOL := FALSE; (*gasmixer 1 - STATE: Warning*)
	bGM2_EnableOperation : BOOL := FALSE; (*gasmixer 2 - enable operation*)
	bGM2_EnableVoltage : BOOL := FALSE; (*gasmixer 2 - enable voltage*)
	bGM2_Error : BOOL := FALSE; (*gasmixer 2 - STATE: Error*)
	bGM2_OperationEnable : BOOL := FALSE; (*gasmixer 2 - STATE: operation enable*)
	bGM2_ReadyToSwitchOn : BOOL := FALSE; (*gasmixer 2 - STATE: ready to switch on*)
	bGM2_ResetError : BOOL := FALSE; (*gasmixer 2 - Reset Error*)
	bGM2_ResetWarning : BOOL := FALSE; (*gasmixer 2 - Reset Warning*)
	bGM2_SetRef : BOOL := TRUE; (*gasmixer 2 - COMMAND: Set Reference*)
	bGM2_SwitchedOn : BOOL := FALSE; (*gasmixer 2 - STATE: switched on*)
	bGM2_SwitchOn : BOOL := FALSE; (*gasmixer 2 - switch on*)
	bGM2_SwitchOnDisabled : BOOL := TRUE; (*gasmixer 2 - STATE: switch on disabled*)
	bGM2_TargetReached : BOOL := FALSE; (*gasmixer 2 - STATE: targed reached*)
	bGM2_Warning : BOOL := FALSE; (*gasmixer 2 - STATE: Warning*)
	rCnt_GM1_SumError : REAL := 0.0; (*gasmixer 1 - counter for position sum error *)
	rCnt_GM2_SumError : REAL := 0.0; (*gasmixer 2 - counter for position sum error *)
	rGM1_MStepRange : REAL := 0.0; (*gasmixer 1 - traversing range [Microsteps]*)
	rGM2_MStepRange : REAL := 0.0; (*gasmixer 2 - traversing range [Microsteps]*)
	rPos_Act_GM1_Norm : REAL := 0.0; (*normed actual gasmixer 1 position from SM1426 [%]*)
	rPos_Act_GM2_Norm : REAL := 0.0; (*normed actual gasmixer 2 position from SM1426 [%]*)
	rPos_GM1_AvgError_Norm : REAL := 0.0; (*gasmixer 1 - normed average position error [%]*)
	rPos_GM1_SumError_Norm : REAL := 0.0; (*gasmixer 1 - normed position sum error [%]*)
	rPos_GM2_AvgError_Norm : REAL := 0.0; (*gasmixer 2 - normed average position error [%]*)
	rPos_GM2_SumError_Norm : REAL := 0.0; (*gasmixer 2 - normed position sum error [%]*)
	xBITtoWD_GM1 : BITtoWD := (0); (*FuB convert Bits to Word*)
	xBITtoWD_GM2 : BITtoWD := (0); (*FuB convert Bits to Word*)
	xTON_GM1_Err : TON := (0); (*FuB*)
	xTON_GM2_Err : TON := (0); (*FuB*)
	xTON_Referencing : TON := (0); (*FuB*)
	xWDtoBIT_GM1 : WDtoBIT := (0); (*FuB convert Word to Bits *)
	xWDtoBIT_GM2 : WDtoBIT := (0); (*FuB convert Word to Bits *)
END_VAR
```

### Program Logical/Gasmixer/Spec_GM (IEC, version 4.05.1) - + special gases mixer

- Spec_GMCyclic.st (not readable text: treated as protected, skipped)

- Spec_GMInit.st (not readable text: treated as protected, skipped)

#### Spec_GM.var
```iecst
VAR
	ss1StepperActPos : INT;
	ss2StepperActPos : INT;
	ss3StepperActPos : INT;
	ssGdr3mmRatedPos : INT;
	ssLdr1mmKollAbst : INT;
	ssLdr1mmRatedPos : INT;
	ssLdr2mmKollAbst : INT;
	ssLdr2mmRatedPos : INT;
	usGdr3mm : UINT;
	usLdr1mm : UINT;
	usLdr2mm : UINT;
	usLdrRel2 : UINT;
	usStepperRatedPos : UINT;
	usRefCounter : UINT;
	usLdr1mmActPosStep : UINT;
	usLdr2mmActPosStep : UINT;
	usGdr3mmActPosStep : UINT;
	TimeBasedOnOff_Stepper1 : TimeBasedOnOff;
	LCCounter_0 : LCCounter;
	TimeBasedOnOff_Stepper2 : TimeBasedOnOff;
	TimeBasedOnOff_Stepper3 : TimeBasedOnOff;
	us2StepperStatus : UINT;
	us1StepperStatus : UINT;
	us3StepperStatus : UINT;
	bInitGo : BOOL;
	TON_Koll : TON;
	TON_Ref : TON;
	ss2EncPosOld : INT;
	ss3EncPosOld : INT;
	TON_ChkDelay : TON;
	TON_Stepper1 : TON;
	TON_Stepper2 : TON;
	TON_Stepper3 : TON;
	TON_RefTime : TON;
	ss1EncPosOld : INT;
	ssGdr3mmActPos : INT;
	TON_SecondTick : TON;
	TON_Stepper2Corr : TON;
	TON_Stepper1Corr : TON;
	TON_Stepper3Corr : TON;
	ssLdr2mmActPos : INT;
	ssLdr1mmActPos : INT;
	usWait : UINT;
	ssPowerOffset1 : INT;
	ssPowerOffset2 : INT;
	ssPowerFactor : INT;
	ucCount : USINT;
	ss1EncPos_Old : INT;
	ss2EncPos_Old : INT;
	ss3EncPos_Old : INT;
	sl1EncPos : DINT;
	sl2EncPos : DINT;
	sl3EncPos : DINT;
	b1StepperDn : BOOL;
	b1StepperUp : BOOL;
	b2StepperDn : BOOL;
	b2StepperUp : BOOL;
	b3StepperDn : BOOL;
	b3StepperUp : BOOL;
	bEncReset : BOOL;
	bGmKoll : BOOL;
	bRefFail : BOOL;
	LeanoxM : BOOL;
	usFaultReason : UINT;
	usKollStatus : UINT;
	usRefStatus : UINT;
	usRefTimes : UINT;
	rP_Act : REAL;
	rP_Set : REAL;
	LdrVoll : ARRAY[0..4] OF UINT;
	OfLdrLl : ARRAY[0..4] OF UINT;
	OfLdrNp : ARRAY[0..4] OF UINT;
	OfLdrSt : ARRAY[0..4] OF UINT;
	ss1EncPos : INT;
	ss1StepRat : INT;
	ss2EncPos : INT;
	ss2StepRat : INT;
	ss3EncPos : INT;
	ss3StepRat : INT;
	rP_Leanox_Act_SP : REAL := 0.0;
END_VAR
```

### Program Logical/Gasmixer/MsgGM (IEC, version 4.01.0) - Alarms generation

#### MsgGMCyclic.st
```iecst
(*******************************************************************************
Msg_GM	 			 alarms generation MM_GasMixer

This code is confidential and proprietary to the INNIO Company.
It may not be used in any form, or reproduced in any manner,
without written permission of the INNIO Company.
Copyright, INNIO Company, 2019

Customized modifications: -
------------------------

History:
-------
V03.99.00.00	23.01.2013	Tinello		new
				27.05.2013	lettenb.	reset OUT_xx.txx2AB.bGnlTripx changed
V04.01.00.00	13.06.2014	Weitzer		add bit for special gasmixer trip 1083
V04.05.00.00	22.01.2018	Tinello		Release Module added

Instructions for use:
--------------------
1) declare alarm with function block "Alm"
	declare buffert alarm bit bMsg<message number>

2) use template to create a new alarm,
   substitue 0000 by alarm number and make settings:

	xMsg0000.Enable		:=	TRUE;		enable/disable alarm
	xMsg0000.Set		:=	FALSE;		alarm set condition
	xMsg0000.PT			:=	T#0s;		alarm delay time
	xMsg0000.Prio		:=	1;			alarm priority: 1-3 = trip, 4 = warning
	xMsg0000.RiskClass	:=	3;			risk class for remote alarm reset
	xMsg0000.Reset		:=	FALSE;		FALSE: for all standard alarms	prio 1,2,3 and warnings prio 4
										TRUE : for autoreset alarms

	bMsg0000			:=	xMsg0000.Q;	connect buffert alarm bit for VIS and control

3)  expand INIT

3)	include datapoint into OPC configuration for vis

Outstandings:
------------
(*******************************************************************************)
PROGRAM _CYCLIC

	(* reset general trip *)
	OUT_GM.tGM2AB.bGnlTrip1		:=	FALSE;
	OUT_GM.tGM2AB.bGnlTrip2		:=	FALSE;
	OUT_GM.tGM2AB.bGnlTrip3		:=	FALSE;
	OUT_GM.tGM2AB.bGnlWarning	:=	FALSE;
	OUT_GM.tGM2AB.bTriptype1	:=	FALSE;
	OUT_GM.tGM2AB.bTriptype2	:=	FALSE;
	OUT_GM.tGM2AB.bTriptype3	:=	FALSE;

	(*---------------------------------------------------------------------------*)
	(* A1083 error gasmixer control *)
	xMsg1083.Enable	   	:= bRelModul_ParaSetupOk;
	xMsg1083.Set       	:= (bErrGM_Ctr OR bErrSGM_Ctr) AND NOT IN_GM.bLeanox_Active AND bOMSS_MAT;
	xMsg1083.PT		   	:= T#0s;
	xMsg1083.Prio	   	:= 2;
	xMsg1083.RiskClass 	:= 3;
	xMsg1083.Reset	   	:= FALSE;
	xMsg1083();
	MM2VIS.bMsg1083		:= xMsg1083.Q;

	(* W2086 measuring signal failure gasmixer position *)
	xMsg2086.Enable	   	:= TRUE;
	xMsg2086.Set       	:= bErrMsGM_Pos;
	xMsg2086.PT		   	:= T#0s;
	xMsg2086.Prio	   	:= 4;
	xMsg2086.RiskClass 	:= 4;
	xMsg2086.Reset	   	:= FALSE;
	xMsg2086();
	MM2VIS.bMsg2086		:= xMsg2086.Q;

	(*---------------------------------------------------------------------------*)
	(* operating messages > AMM *)

	(* B template
	xMsg.Enable		:=	TRUE;
	xMsg.Set		:=	bBool;
	xMsg.Reset		:=	TRUE;
	xMsg();
	MM2VIS.bMsg		:=	xMsg.Q;	*)

	(*---------------------------------------------------------------------------*)
	(* general alarms for further module operations *)
	bGnlTrip1 	:= OUT_GM.tGM2AB.bGnlTrip1 		OR IN_GM.tAB2GM.bGnlTrip1;
	bGnlTrip2 	:= OUT_GM.tGM2AB.bGnlTrip2 		OR IN_GM.tAB2GM.bGnlTrip2;
	bGnlTrip3 	:= OUT_GM.tGM2AB.bGnlTrip3 		OR IN_GM.tAB2GM.bGnlTrip3;
	bGnlWarning := OUT_GM.tGM2AB.bGnlWarning 	OR IN_GM.tAB2GM.bGnlWarning;
	bGnlTrip	:= bGnlTrip1 OR bGnlTrip2 OR bGnlTrip3;

(*******************************************************************************)
END_PROGRAM
```

#### MsgGMInit.st - Cyclic code
```iecst
(*******************************************************************************
Msg_GM	 			 alarms generation MM_GasMixer

This code is confidential and proprietary to the INNIO Company.
It may not be used in any form, or reproduced in any manner,
without written permission of the INNIO Company.
Copyright, INNIO Company, 2019

Customized modifications: -
------------------------

History:
-------
V03.99.00.00	23.01.2013 	Tinello 	new

Instructions for use:
--------------------
1) declare alarm with function block "Msg"

2) use template to create a new alarm, substitue 0000 by message number:

	xMsg0000.Num		:=	0000;					alarm number
	xMsg0000.AmmSysAdr	:=  iAdrAmmBase2MM;			do not change
	xMsg0000.AmmOutAdr	:=  iAdrMM2AmmBase;			do not change

3) 	set alarm number

Outstandings:
------------
(*******************************************************************************)
PROGRAM _INIT

	iAdrAmmBase2MM		:= ADR(IN_GM.tAB2GM);
	iAdrMM2AmmBase		:= ADR(OUT_GM.tGM2AB);

	(*---------------------------------------------------------------------------*)

	xMsg1083.Num		:= 1083;
	xMsg1083.AmmInAdr	:= iAdrAmmBase2MM;
	xMsg1083.AmmOutAdr	:= iAdrMM2AmmBase;

	xMsg2086.Num		:= 2086;
	xMsg2086.AmmInAdr	:= iAdrAmmBase2MM;
	xMsg2086.AmmOutAdr	:= iAdrMM2AmmBase;

END_PROGRAM
```

#### MsgGM.var
```iecst
VAR
	iAdrAmmBase2MM : UDINT;
	iAdrMM2AmmBase : UDINT;
	xMsg1083 : Msg; (*error gasmixer control*)
	xMsg2086 : Msg; (*measuring signal failure gasmixer position*)
END_VAR
```

### Program Logical/Gasmixer/ParGM (IEC, version 4.06.0) - + save parameters

- perm_par.st (not readable text: treated as protected, skipped)
